// TIA Portal project "LCR 01-001" (V14)
// Atualização de hardware e software, melhorais na estrela de frasco

(* hardware
DEVICE "S7-1200 station_1"  S7-1200 Station
   slot 0: "Rack_0"  S7-1200 Rack  Rack  V1.0
   slot 1: "PLC_1"  CPU 1212C DC/DC/DC  6ES7 212-1AE40-0XB0  V4.2
   slot 3: "DQ 4x24VDC_1"  DQ4 signal board (200 kHz)  6ES7 222-1BD30-0XB0  V1.0
DEVICE "GSD device_1"  GSD.Device.PN
   slot 0: "Rack"  Rack  V1.0
   slot 0: "16DI"  16DI
   slot 0: "16DO"  16DO
   slot 0: "16DO"  16DO
   slot 0: "8DI"  8DI
   slot 0: "wago-750-375"  750-375 V02.02.xx (FW 05)  750-375  V02.02.xx (05)
      slot 0: "Big Endian (MOTOROLA), Subslot-controlled PROFIenergy"  Big Endian (MOTOROLA), Subslot-controlled PROFIenergy
      slot 1: "Interface"  Interface
         slot 1: "Port 1"  Port 1
         slot 2: "Port 2"  Port 2
   slot 1: "750-1405 16DI_1"  750-1405 16DI  750-1405
   slot 2: "750-1504 16DO_1"  750-1504 16DO  750-1504
   slot 3: "750-1504 16DO_2"  750-1504 16DO  750-1504
   slot 4: "75x-430(/0..-...) 8DI_1"  75x-430(/0..-...) 8DI  75x-430
*)

// ===== PLC "PLC_1"  CPU 1212C DC/DC/DC =====

VAR_GLOBAL   // PLC tag table "Default tag table"
   "Sensor home Platô" AT %I0.0 : Bool;
   "Sensor home Estrela" AT %I0.1 : Bool;
   "Sensor home Dosador" AT %I0.2 : Bool;
   "Sensor Limite superior Dosador" AT %I0.3 : Bool;
   "Sensor DR valvula Dosador" AT %I0.4 : Bool;
   "Sensor EQ valvula Dosador" AT %I0.5 : Bool;
   "Sensor home trans manipulador" AT %I0.6 : Bool;
   "Sensor CNT frasco dosador" AT %I0.7 : Bool;
   "Sensor CNT tampa rosqueador" AT %I1.0 : Bool;
   "Sensor canaleta de frasco" AT %I1.1 : Bool;
   "Sensor direito canaleta de tampa" AT %I1.2 : Bool;
   "Sensor esquerdo canaleta de tampa" AT %I1.3 : Bool;
   "Sensor cilindro manipulador" AT %I1.4 : Bool;
   "Sensor cilindro rosqueador" AT %I1.5 : Bool;
   "Sensor visão artificial" AT %I1.6 : Bool;
   "Sobrecarga_manipulador" AT %I1.7 : Bool;
   "Emergência" AT %I2.0 : Bool;
   "Automatico" AT %I2.1 : Bool;
   "Liga" AT %I2.2 : Bool;
   "Desliga" AT %I2.3 : Bool;
   "Reset falhas" AT %I2.4 : Bool;
   "Ativoalarmeplatô" AT %I2.5 : Bool;
   "Ativoalarmeestrela" AT %I2.6 : Bool;
   "Ativoalarmedosador" AT %I2.7 : Bool;
   "Entrada analogica" AT %IW64 : Word;
   "Sensor pressão" AT %ID200 : DWord;
   "AUX" AT %ID204 : Real;
   "CONTROLE" AT %ID208 : Real;
   "Alarme_disjunto_wago" AT %I3.0 : Bool;
   "Alvo_atingido_torque" AT %I3.1 : Bool;
   "Sensor_detector_inspeção" AT %I3.2 : Bool;
   "Sensor_CNT_manipulador" AT %I3.3 : Bool;
   "Platô_Pulse" AT %Q4.0 : Bool;
   "Platô_Direction" AT %Q4.1 : Bool;
   "Estrela_Pulse" AT %Q4.2 : Bool;
   "Estrela_Direction" AT %Q4.3 : Bool;
   "Envase_Pulse" AT %Q0.0 : Bool;
   "Envase_Direction" AT %Q0.1 : Bool;
   "Trans manipulador_Pulse" AT %Q0.2 : Bool;
   "Trans manipulador_Direction" AT %Q0.3 : Bool;
   "Smart_camera" AT %Q0.4 : Bool;
   "reservado(5)" AT %Q0.5 : Bool;
   "Gira posicinador direito tampa" AT %Q1.0 : Bool;
   "Home posicionador direito" AT %Q1.1 : Bool;
   "Gira posicionador esquerdo" AT %Q1.2 : Bool;
   "Home posicionador esquerdo" AT %Q1.3 : Bool;
   "Rosqueador aplicação tampa" AT %Q1.4 : Bool;
   "Continuo_Rosqueador" AT %Q1.5 : Bool;
   "Solenoide Rosqueador tampa" AT %Q1.6 : Bool;
   "Solenoide Manipulador tampa" AT %Q1.7 : Bool;
   "Solenoide empurrador tampa" AT %Q2.0 : Bool;
   "Solenoide valvula dosagem" AT %Q2.1 : Bool;
   "Solenoide frasco reprovado" AT %Q2.2 : Bool;
   "Válvula vacuo Pegador 1" AT %Q2.3 : Bool;
   "Válvula vacuo pegador 2" AT %Q2.4 : Bool;
   "Válvula vacuo estrela" AT %Q2.5 : Bool;
   "Válvula sopro pegador 1" AT %Q2.6 : Bool;
   "Válvula sopro pegador 2" AT %Q2.7 : Bool;
   "Válvula sopro canleta dire" AT %Q5.0 : Bool;
   "Válvula sopro canaleta esque" AT %Q5.1 : Bool;
   "Habilita alimentadores" AT %Q5.2 : Bool;
   "Alimentador de frasco" AT %Q5.3 : Bool;
   "Alimentador de tampa" AT %Q5.4 : Bool;
   "LED máquina on" AT %Q5.5 : Bool;
   "LED alarme" AT %Q5.6 : Bool;
   "LED máquina off" AT %Q5.7 : Bool;
   "Reset disjuntor eletrônico" AT %Q6.0 : Bool;
   "Reset servodrives" AT %Q6.1 : Bool;
   "Jog platô avança SV" AT %Q6.2 : Bool;
   "Jog platô recuo SV" AT %Q6.3 : Bool;
   "Jog estrela avança SV" AT %Q6.4 : Bool;
   "Jog estrela recuo SV" AT %Q6.5 : Bool;
   "Sensor_detector" AT %Q6.6 : Bool;
   "Tag_1" AT %Q6.7 : Bool;
   "System_Byte" AT %MB1 : Byte;
   "FirstScan" AT %M1.0 : Bool;
   "DiagStatusUpdate" AT %M1.1 : Bool;
   "AlwaysTRUE" AT %M1.2 : Bool;
   "AlwaysFALSE" AT %M1.3 : Bool;
   "Clock_Byte" AT %MB0 : Byte;
   "Clock_10Hz" AT %M0.0 : Bool;
   "Clock_5Hz" AT %M0.1 : Bool;
   "Clock_2.5Hz" AT %M0.2 : Bool;
   "Clock_2Hz" AT %M0.3 : Bool;
   "Clock_1.25Hz" AT %M0.4 : Bool;
   "Clock_1Hz" AT %M0.5 : Bool;
   "Clock_0.625Hz" AT %M0.6 : Bool;
   "Clock_0.5Hz" AT %M0.7 : Bool;
   "Alarme alimentador desligado" AT %M2.1 : Bool;
   "Canaletas de tampa cheia" AT %M2.2 : Bool;
   "Canaleta de tamapa vasia" AT %M2.3 : Bool;
   "Alarme falta frasco" AT %M2.4 : Bool;
   "Alarme falta tampa" AT %M2.5 : Bool;
   "Liga Máquina" AT %M2.0 : Bool;
   "Pulso  deslocamento trans" AT %M2.6 : Bool;
   "Platô em deslocamento" AT %M2.7 : Bool;
   "Platô_Alvo atingido" AT %M3.0 : Bool;
   "Estrela em deslocamento" AT %M3.1 : Bool;
   "Estrela_Alvo atingido" AT %M3.2 : Bool;
   "Envase em deslocamento" AT %M3.3 : Bool;
   "Envase_Alvo atingido" AT %M3.4 : Bool;
   "Manipulador em deslocamento" AT %M3.5 : Bool;
   "Manipulador_Alvo atingido" AT %M3.6 : Bool;
   "Falha platô" AT %M3.7 : Bool;
   "Falha etrela" AT %M4.0 : Bool;
   "Falha  envase" AT %M4.1 : Bool;
   "Falha manipu" AT %M4.2 : Bool;
   "Pulso deslocamento envase" AT %M4.3 : Bool;
   "Iniciaenvase" AT %M4.4 : Bool;
   "Iniciaenchimento" AT %M4.5 : Bool;
   "Envase_echimento alvo atingido" AT %M4.6 : Bool;
   "Envase_enchimento em deslocamento" AT %M4.7 : Bool;
   "Avança manipulador" AT %M5.0 : Bool;
   "Recuo manipulador" AT %M5.1 : Bool;
   "Set on Home platô" AT %M5.2 : Bool;
   "Set on Home estrela" AT %M5.3 : Bool;
   "Set on Home envase" AT %M5.4 : Bool;
   "Set on Home mani" AT %M5.5 : Bool;
   "Rqs_SaveReceita" AT %M6.0 : Bool;
   "Download_receita" AT %M6.1 : Bool;
   "Pulso_valavula_dosagem" AT %M6.2 : Bool;
   "Atenção" AT %M6.3 : Bool;
   "Estações_Nsincronizada" AT %M6.4 : Bool;
   "Estçoes_emhome" AT %M6.5 : Bool;
   "Bit_on" AT %M6.6 : Bool;
   "Startup_emergência" AT %M6.7 : Bool;
   "Alvo_atingidoavançoMN" AT %M7.0 : Bool;
   "Alvo_atingidorecuoMN" AT %M7.1 : Bool;
   "Deslocamento_avançoMN" AT %M7.2 : Bool;
   "Deslocamento_recuoMN" AT %M7.3 : Bool;
   "Alarme_manutenção" AT %M7.4 : Bool;
   "Status_deslocamento_rosqueador" AT %M7.5 : Bool;
   "Erro" AT %MW8 : Int;
END_VAR

TYPE "UDT_Dados_máquina"
VERSION : 0.1
   STRUCT
      Qauntidade_partida : DInt;
      Maquina_ligadahoras : DInt;
      Maquina_ligadaminutos : DInt;
      Proxima_manutenção : DInt := 0;
      Preset_manutenção : DInt;
      Salva_proximamanutenção : Bool;
   END_STRUCT;
END_TYPE

DATA_BLOCK "Start stop Machine_DB"   // DB25
{ S7_Optimized_Access := 'TRUE' }
VERSION : 0.1
// stored: InstanceOfName Start stop Machine
"Start stop Machine"
BEGIN
END_DATA_BLOCK

DATA_BLOCK "Parâmetros platô estrela"   // DB26
{ S7_Optimized_Access := 'FALSE' }
VERSION : 0.1
   VAR
      "Habilita servo drive P" : Bool;
      "Habilita Servo drive E" : Bool;
      "Habilita rampa AC/DC P" : Bool;
      "Habilita rampa AC/Dc E" : Bool;
      "Home platô" : Bool;
      "Home estrela" : Bool;
      "Jog Avanço P" : Bool;
      "Jog Recuo P" : Bool;
      "Jog avanço E" : Bool;
      "Jog recuo E" : Bool;
      "Jog avanço teste" : Bool;
      "Reset posição" : Real;
      "Jog recuo teste" : Bool;
      "Rampa aceleração" : Int;
      "Rampa desaceleração" : Int;
      "Velocidade máquina" : Int;
      "Fino home platô" : Int;
      "Fino home estrela" : Int;
      "Contador de frasco" : Int;
      Velocidadereal : Real;
      "Rampaaceleração Real" : Real;
      RampadesaceleraçãoReal : Real;
      "Fino home platô Real" : Real;
      "Fino Home estrela Real" : Real;
      "Ativa parametro" : Bool;
      "Intervalo X" : Real;
      "RampaREAL AC" : Real;
      "RampaREAL DC" : Real;
      "Home platô ON" : Bool;
      "Home estrela ON" : Bool;
      "Vacuo estrela" : Bool;
      "posição atual" : Real;
      Ganho_RPM_estrela : Real;
      Posição_atualP : Int;
      "Offset home" : Real;
      Loadparametro : Bool;
   END_VAR
BEGIN
END_DATA_BLOCK

DATA_BLOCK "Alarme_Bit"   // DB27
{ S7_Optimized_Access := 'FALSE' }
VERSION : 0.1
   VAR
      Status_sincrinizamos : Bool;
      Emergência : Bool;
      "Servo drive platõ em flha" : Bool;
      "Servo drive estrela em flha" : Bool;
      "Servo drive dosador em falha" : Bool;
      "alimentadores desligado" : Bool;
      "Alarme falta de frasco" : Bool;
      "Alrme falta de tampa" : Bool;
      "Falha instrução platô" : Bool;
      "Falha Instrução etrela" : Bool;
      "Falha instrução envase" : Bool;
      "Falha instrução manipu" : Bool;
      Falha_arcomprimido : Bool;
      Falha_Valvuladosagen : Bool;
      Falha_manipulador : Bool;
      Limite_horas : Bool;
      Sobrecarga_manipulador : Bool;
      Falha_subida_rosqueador : Bool;
      Falha_recuo_dosador : Bool;
      Falha_sensor_valvula : Bool;
   END_VAR
BEGIN
END_DATA_BLOCK

DATA_BLOCK "Parâmetros de envase"   // DB28
{ S7_Optimized_Access := 'FALSE' }
VERSION : 0.1
   VAR
      "Habilita Servo drive D" : Bool := FALSE;
      "Habilita rampa AC/DC D" : Bool := FALSE;
      "Home dosador" : Bool := FALSE;
      "Jog avanço D" : Bool := FALSE;
      "Jog recuo D" : Bool := FALSE;
      "Coreção ml" : Int := 0;
      "Rampa acelreção D" : Int := 0;
      "Rampa desaceleração D" : Int := 0;
      "Velocidade envase" : Int := 0;
      "Velocidade enchimento" : Int := 0;
      Deslocamento : Real;
      Deslocamento_1 : Real := 0.0;
      "Velocidade envase_1" : Real := 0.0;
      "Velcidade envase_2" : Real;
      Posiçãoatual : Real;
      AtivaparametrosRampa : Bool;
      "Velocidade enchimento_1" : Real;
      "Velocidade enchimento_2" : Real;
      Ramp_AC1 : Real;
      Ramp_AC2 : Real;
      Ramp_DC1 : Real;
      Ramp_DC2 : Real;
      "Home envase ON" : Bool;
      Atual_posição : Real;
      Atual_posição_scalX : Real;
      Atual_Posição_IHM : Int;
      Status_lavgem : Bool;
   END_VAR
BEGIN
END_DATA_BLOCK

DATA_BLOCK "Parâmetros rosqueador"   // DB29
{ S7_Optimized_Access := 'FALSE' }
VERSION : 0.1
   VAR
      "Desce rosqueador" : Bool;
      "Ciclo de fechamento" : Bool;
      Inter_conti : Bool;
      "Tempo deslocame_real" : Time;
      "Tempo deslocamento" : Time;
      Inicio_torque : Time;
   END_VAR
BEGIN
END_DATA_BLOCK

DATA_BLOCK "Parâmetros alimentadores_1"   // DB30
{ S7_Optimized_Access := 'FALSE' }
VERSION : 0.1
   VAR
      "Habilita frasco" : Bool;
      "Habilita tampa" : Bool;
      "ON alarme falat frasco" : Bool;
      "ON alarme falta tampa" : Bool;
      "Liga alimentadores" : Bool;
      "Retardo liga frasco" : DInt;
      "Retardo desliga frasco" : DInt;
      "Retardo liga tampa" : DInt;
      "Retardo desliga tampa" : DInt;
      "Retardo sopro D" : DInt;
      "Retardo sopro E" : DInt;
      "Retardo falta de frasco" : DInt;
      "Retardo falta de tampa" : DInt;
      Aux_realtampa : DInt;
      Aux_realfrasco : DInt;
      "Ar comprimido" : Int;
      Real_timerTampa : Int;
      Real_timerfrasco : Int;
   END_VAR
BEGIN
END_DATA_BLOCK

DATA_BLOCK "Parâmetros manipuladpor"   // DB31
{ S7_Optimized_Access := 'FALSE' }
VERSION : 0.1
   VAR
      "Habilita STR8" : Bool;
      "Habilita rampa AC/DC" : Bool;
      "Home manipulador" : Bool;
      "Jog avanço mani" : Bool;
      "Jog recuo mani" : Bool;
      "Home posici direito" : Bool;
      "Home posici esquerdo" : Bool;
      "Rampa aceleração mani" : Int;
      "Rampa desaceleração mani" : Int;
      "RPM manipulador" : Int;
      "RPM manipulador_1" : Real;
      "RPM manipulador_2" : Real;
      "Ramp AC_1" : Real;
      "Ramp AC_2" : Real;
      "Ramp DC_1" : Real;
      "Ramp DC_2" : Real;
      "ativa parametro" : Bool;
      "Posição atual_1" : Real;
      "Posição atual" : Int;
      "Home mani ON" : Bool;
      Tampa_frasco : Bool;
   END_VAR
BEGIN
END_DATA_BLOCK

DATA_BLOCK "Parâmetros de produção"   // DB32
{ S7_Optimized_Access := 'FALSE' }
VERSION : 0.1
   VAR
      "Habilita contador de lote" : Bool;
      Rejeito : Bool;
      Teste_Sensor : Bool;
      Rest_produção : Bool;
      "Peças por minuto" : DInt;
      "Total por minuto" : DInt;
      "Total por minuto_1" : Int;
      TImer_1 : Time;
      Timer_2 : Time;
      AUX_produção : Int;
   END_VAR
BEGIN
END_DATA_BLOCK

DATA_BLOCK "DB_pulso"   // DB38
{ S7_Optimized_Access := 'TRUE' }
VERSION : 0.1
   VAR
      Manual : Bool;
      Pulso_PL_ES : Array[0..12] of Bool;
      Pulso_EV : Array[0..20] of Bool;
      Pulso_MN : Array[0..25] of Bool;
      Pulso_RQ : Array[0..10] of Bool;
      Pulso_ALM : Array[0..20] of Bool;
      Pulso_receita : Array[0..5] of Bool;
      Pulso_alarme : Array[0..20] of Bool;
      Controle_produção : Array[0..20] of Bool;
      Startup : Array[0..20] of Bool;
      UDT_máquina : Array[0..5] of Bool;
   END_VAR
BEGIN
END_DATA_BLOCK

DATA_BLOCK "Comando transmissão_DB"   // DB43
{ S7_Optimized_Access := 'TRUE' }
VERSION : 0.1
// stored: InstanceOfName Comando transmissão
"Comando transmissão"
BEGIN
END_DATA_BLOCK

DATA_BLOCK "Comando valvula dosador_DB"   // DB48
{ S7_Optimized_Access := 'TRUE' }
VERSION : 0.1
// stored: InstanceOfName Comando valvula dosador
"Comando valvula dosador"
BEGIN
END_DATA_BLOCK

DATA_BLOCK "Controle manipulador_DB"   // DB51
{ S7_Optimized_Access := 'TRUE' }
VERSION : 0.1
// stored: InstanceOfName Controle manipulador
"Controle manipulador"
BEGIN
END_DATA_BLOCK

DATA_BLOCK "DB_UDT_dadosMáqquin"   // DB53
{ S7_Optimized_Access := 'FALSE' }
VERSION : 0.1
   VAR
      Plc_DT_atual : DTL;
      Retorvalor : Int;
      Máquina : Array[0..0] of "UDT_Dados_máquina";
      Aux_preset : Int;
      Aux_horas : Int;
      Aux_minuto : Int;
      Aux_partida : Int;
   END_VAR
BEGIN
END_DATA_BLOCK

DATA_BLOCK "DB_Receitas"   // DB55
{ S7_Optimized_Access := 'FALSE' }
VERSION : 0.1
   VAR
      Receita : Array[0..20] of Word;
      Rqs_DownloadReceita : Bool;
      Rqs_SaveReceita : Bool;
   END_VAR
BEGIN
END_DATA_BLOCK

DATA_BLOCK "Parâmetros_IHM"   // DB56
{ S7_Optimized_Access := 'FALSE' }
VERSION : 0.1
   VAR
      Int_1 : Int;
      Int_2 : Int;
      Int_3 : Int;
      Int_4 : Int;
      Int_5 : Int;
      Int_6 : Int;
      Int_7 : Int;
      Int_8 : Int;
      Int_9 : Int;
      Int_10 : Int;
      Int_11 : Int;
      Int_12 : Int;
      Int_13 : Int;
      Int_14 : Int;
      Int_15 : Int;
      Int_16 : Int;
      Int_17 : Int;
      Int_18 : Int;
      Int_19 : Int;
      Int_20 : Int;
      Int_21 : Int;
      Int_22 : Int;
      Int_23 : Int;
      Int_24 : Int;
      Int_25 : Int;
      Int_26 : Int;
      Int_27 : Int;
      Int_28 : Int;
      Int_29 : Int;
      Int_30 : Int;
      Int_31 : Int;
      Int_32 : Int;
      Int_33 : Int;
      Int_34 : Int;
      Int_35 : Int;
      Int_36 : Int;
      Int_37 : Int;
      Int_38 : Int;
      Int_39 : Int;
      Int_40 : Int;
      DBW_0 : Word;
   END_VAR
BEGIN
END_DATA_BLOCK

DATA_BLOCK "Parâmetros_BooL_IHM"   // DB57
{ S7_Optimized_Access := 'FALSE' }
VERSION : 0.1
   VAR
      St001 : Bool;
      St002 : Bool;
      St003 : Bool;
      St004 : Bool;
      St005 : Bool;
      St006 : Bool;
      St007 : Bool;
      St008 : Bool;
      St009 : Bool;
      St010 : Bool;
      St011 : Bool;
      St012 : Bool;
      St013 : Bool;
      St014 : Bool;
      St015 : Bool;
      St016 : Bool;
      St017 : Bool;
      St018 : Bool;
      St019 : Bool;
      St020 : Bool;
      Status_W0 : Int;
      Status_W1 : Int;
   END_VAR
BEGIN
END_DATA_BLOCK

DATA_BLOCK "Rosqueador_tampa_DB"   // DB59
{ S7_Optimized_Access := 'TRUE' }
VERSION : 0.1
// stored: InstanceOfName Rosqueador_tampa
"Rosqueador_tampa"
BEGIN
END_DATA_BLOCK

DATA_BLOCK "Alarme_mensagen"   // DB60
{ S7_Optimized_Access := 'FALSE' }
VERSION : 0.1
   VAR
      Mensagen_1 : Array[0..15] of Word;
   END_VAR
BEGIN
END_DATA_BLOCK

DATA_BLOCK "DB_Startup"   // DB68
{ S7_Optimized_Access := 'TRUE' }
VERSION : 0.1
   VAR
      Stsrtup : Array[0..10] of Bool;
   END_VAR
BEGIN
END_DATA_BLOCK

DATA_BLOCK "Presença"   // DB72
{ S7_Optimized_Access := 'FALSE' }
VERSION : 0.1
   VAR
      Presenca_08 : Bool;
      Presenca_09 : Bool;
      Presenca_10 : Bool;
      Presenca_11 : Bool;
      Presenca_12 : Bool;
      Presenca_13 : Bool;
      Presenca_14 : Bool;
      Presenca_15 : Bool;
      Presenca_00 : Bool;
      Presenca_01 : Bool;
      Presenca_02 : Bool;
      Presenca_03 : Bool;
      Presenca_04 : Bool;
      Presenca_05 : Bool;
      Presenca_06 : Bool;
      Presenca_07 : Bool;
   END_VAR
BEGIN
END_DATA_BLOCK

// folder: System blocks/Program resources

DATA_BLOCK "IEC_Timer_0_DB"   // DB33
{ S7_Optimized_Access := 'TRUE' }
AUTHOR : Simatic
FAMILY : IEC
NAME : IEC_TMR
VERSION : 1.0
// stored: InstanceOfName IEC_TIMER
"IEC_TIMER"
BEGIN
END_DATA_BLOCK

DATA_BLOCK "IEC_Timer_0_DB_1"   // DB34
{ S7_Optimized_Access := 'TRUE' }
AUTHOR : Simatic
FAMILY : IEC
NAME : IEC_TMR
VERSION : 1.0
// stored: InstanceOfName IEC_TIMER
"IEC_TIMER"
BEGIN
END_DATA_BLOCK

DATA_BLOCK "IEC_Timer_0_DB_2"   // DB35
{ S7_Optimized_Access := 'TRUE' }
AUTHOR : Simatic
FAMILY : IEC
NAME : IEC_TMR
VERSION : 1.0
// stored: InstanceOfName IEC_TIMER
"IEC_TIMER"
BEGIN
END_DATA_BLOCK

DATA_BLOCK "IEC_Timer_0_DB_3"   // DB36
{ S7_Optimized_Access := 'TRUE' }
AUTHOR : Simatic
FAMILY : IEC
NAME : IEC_TMR
VERSION : 1.0
// stored: InstanceOfName IEC_TIMER
"IEC_TIMER"
BEGIN
END_DATA_BLOCK

DATA_BLOCK "IEC_Timer_0_DB_4"   // DB37
{ S7_Optimized_Access := 'TRUE' }
AUTHOR : Simatic
FAMILY : IEC
NAME : IEC_TMR
VERSION : 1.0
// stored: InstanceOfName IEC_TIMER
"IEC_TIMER"
BEGIN
END_DATA_BLOCK

DATA_BLOCK "IEC_Timer_0_DB_5"   // DB39
{ S7_Optimized_Access := 'TRUE' }
AUTHOR : Simatic
FAMILY : IEC
NAME : IEC_TMR
VERSION : 1.0
// stored: InstanceOfName IEC_TIMER
"IEC_TIMER"
BEGIN
END_DATA_BLOCK

DATA_BLOCK "IEC_Timer_0_DB_6"   // DB40
{ S7_Optimized_Access := 'TRUE' }
AUTHOR : Simatic
FAMILY : IEC
NAME : IEC_TMR
VERSION : 1.0
// stored: InstanceOfName IEC_TIMER
"IEC_TIMER"
BEGIN
END_DATA_BLOCK

DATA_BLOCK "IEC_Timer_0_DB_7"   // DB41
{ S7_Optimized_Access := 'TRUE' }
AUTHOR : Simatic
FAMILY : IEC
NAME : IEC_TMR
VERSION : 1.0
// stored: InstanceOfName IEC_TIMER
"IEC_TIMER"
BEGIN
END_DATA_BLOCK

DATA_BLOCK "IEC_Timer_0_DB_8"   // DB42
{ S7_Optimized_Access := 'TRUE' }
AUTHOR : Simatic
FAMILY : IEC
NAME : IEC_TMR
VERSION : 1.0
// stored: InstanceOfName IEC_TIMER
"IEC_TIMER"
BEGIN
END_DATA_BLOCK

DATA_BLOCK "IEC_Timer_0_DB_9"   // DB50
{ S7_Optimized_Access := 'TRUE' }
AUTHOR : Simatic
FAMILY : IEC
NAME : IEC_TMR
VERSION : 1.0
// stored: InstanceOfName IEC_TIMER
"IEC_TIMER"
BEGIN
END_DATA_BLOCK

DATA_BLOCK "IEC_Timer_0_DB_10"   // DB61
{ S7_Optimized_Access := 'TRUE' }
AUTHOR : Simatic
FAMILY : IEC
NAME : IEC_TMR
VERSION : 1.0
// stored: InstanceOfName IEC_TIMER
"IEC_TIMER"
BEGIN
END_DATA_BLOCK

DATA_BLOCK "IEC_Timer_0_DB_11"   // DB62
{ S7_Optimized_Access := 'TRUE' }
AUTHOR : Simatic
FAMILY : IEC
NAME : IEC_TMR
VERSION : 1.0
// stored: InstanceOfName IEC_TIMER
"IEC_TIMER"
BEGIN
END_DATA_BLOCK

DATA_BLOCK "IEC_Timer_0_DB_12"   // DB63
{ S7_Optimized_Access := 'TRUE' }
AUTHOR : Simatic
FAMILY : IEC
NAME : IEC_TMR
VERSION : 1.0
// stored: InstanceOfName IEC_TIMER
"IEC_TIMER"
BEGIN
END_DATA_BLOCK

DATA_BLOCK "IEC_Timer_0_DB_19"   // DB64
{ S7_Optimized_Access := 'TRUE' }
AUTHOR : Simatic
FAMILY : IEC
NAME : IEC_TMR
VERSION : 1.0
// stored: InstanceOfName IEC_TIMER
"IEC_TIMER"
BEGIN
END_DATA_BLOCK

DATA_BLOCK "IEC_Timer_0_DB_13"   // DB65
{ S7_Optimized_Access := 'TRUE' }
AUTHOR : Simatic
FAMILY : IEC
NAME : IEC_TMR
VERSION : 1.0
// stored: InstanceOfName IEC_TIMER
"IEC_TIMER"
BEGIN
END_DATA_BLOCK

DATA_BLOCK "IEC_Timer_0_DB_14"   // DB66
{ S7_Optimized_Access := 'TRUE' }
AUTHOR : Simatic
FAMILY : IEC
NAME : IEC_TMR
VERSION : 1.0
// stored: InstanceOfName IEC_TIMER
"IEC_TIMER"
BEGIN
END_DATA_BLOCK

DATA_BLOCK "IEC_Timer_0_DB_15"   // DB67
{ S7_Optimized_Access := 'TRUE' }
AUTHOR : Simatic
FAMILY : IEC
NAME : IEC_TMR
VERSION : 1.0
// stored: InstanceOfName IEC_TIMER
"IEC_TIMER"
BEGIN
END_DATA_BLOCK

DATA_BLOCK "IEC_Timer_0_DB_16"   // DB69
{ S7_Optimized_Access := 'TRUE' }
AUTHOR : Simatic
FAMILY : IEC
NAME : IEC_TMR
VERSION : 1.0
// stored: InstanceOfName IEC_TIMER
"IEC_TIMER"
BEGIN
END_DATA_BLOCK

DATA_BLOCK "IEC_Timer_0_DB_17"   // DB70
{ S7_Optimized_Access := 'TRUE' }
AUTHOR : Simatic
FAMILY : IEC
NAME : IEC_TMR
VERSION : 1.0
// stored: InstanceOfName IEC_TIMER
"IEC_TIMER"
BEGIN
END_DATA_BLOCK

DATA_BLOCK "IEC_Timer_0_DB_18"   // DB71
{ S7_Optimized_Access := 'TRUE' }
AUTHOR : Simatic
FAMILY : IEC
NAME : IEC_TMR
VERSION : 1.0
// stored: InstanceOfName IEC_TIMER
"IEC_TIMER"
BEGIN
END_DATA_BLOCK

// folder: (top level)

DATA_BLOCK "Platô"   // DB2, Motion_DB
{ S7_Optimized_Access := 'TRUE' }
AUTHOR : SIMATIC
FAMILY : BasicMC
NAME : TO_PosAx
VERSION : 5.0
// stored: InstanceOfName TO_PositioningAxis
"TO_PositioningAxis"
BEGIN
   // Axis.LengthUnitNormalized.Distance = 1005
   // Axis.PositionLimitsMin_AddressCU = %I0.0
   // Axis.DirectionOutputEnabledCU = TRUE
   // Axis.PassiveHomingReferencePointSwitch_AddressCU = %I0.0
   // Axis.HomingReferencePointSwitch_AddressCU = %I0.0
   // Axis.OnlinePtoModeCUEnumValue = PTO (pulse A and direction B)
   // Axis.OnlinePtoModeCU = 16#0000_0002
   // Axis.SelectedChannel2EnumCU = %Q4.1
   // Axis.SelectedChannel1EnumCU = %Q4.0
   // Pulse.MinDeltaDeltaFrequencyCU = 0.004
   // Pulse.MaxDeltaDeltaFrequencyCU = 1.0E+10
   // Pulse.MinDeltaFrequencyCU = 0.005
   // Pulse.MaxDeltaFrequencyCU = 9.5E+9
   // Pulse.MinFrequencyCU = 1.0
   // Pulse.MaxFrequencyCU = 200000.0
   // Pulse.OutputSourceCU = 16#0000_0001
   // Axis.SelectPTO = 0
   // Axis.LengthUnit.LastDistance = 1005
END_DATA_BLOCK

DATA_BLOCK "Estrela"   // DB3, Motion_DB
{ S7_Optimized_Access := 'TRUE' }
AUTHOR : SIMATIC
FAMILY : BasicMC
NAME : TO_PosAx
VERSION : 5.0
// stored: InstanceOfName TO_PositioningAxis
"TO_PositioningAxis"
BEGIN
   // Axis.PositionLimitsMin_AddressCU = %I0.1
   // Axis.PassiveHomingReferencePointSwitch_AddressCU = %I0.1
   // Axis.HomingReferencePointSwitch_AddressCU = %I0.1
   // Axis.LengthUnitNormalized.Distance = 1005
   // Axis.DirectionOutputEnabledCU = TRUE
   // Axis.OnlinePtoModeCUEnumValue = PTO (pulse A and direction B)
   // Axis.OnlinePtoModeCU = 16#0000_0002
   // Axis.SelectedChannel2EnumCU = %Q4.3
   // Axis.SelectedChannel1EnumCU = %Q4.2
   // Pulse.MinDeltaDeltaFrequencyCU = 0.004
   // Pulse.MaxDeltaDeltaFrequencyCU = 1.0E+10
   // Pulse.MinDeltaFrequencyCU = 0.005
   // Pulse.MaxDeltaFrequencyCU = 9.5E+9
   // Pulse.MinFrequencyCU = 1.0
   // Pulse.MaxFrequencyCU = 200000.0
   // Pulse.OutputSourceCU = 16#0000_0001
   // Axis.SelectPTO = 1
   // Axis.OnlinePtoIndexCU = 1
   // Axis.LengthUnit.LastDistance = 1005
END_DATA_BLOCK

DATA_BLOCK "Envase"   // DB4, Motion_DB
{ S7_Optimized_Access := 'TRUE' }
AUTHOR : SIMATIC
FAMILY : BasicMC
NAME : TO_PosAx
VERSION : 5.0
// stored: InstanceOfName TO_PositioningAxis
"TO_PositioningAxis"
BEGIN
   // Axis.PositionLimitsMax_AddressCU = %I0.3
   // Axis.PositionLimitsMin_AddressCU = %I0.2
   // Axis.PassiveHomingReferencePointSwitch_AddressCU = %I0.2
   // Axis.HomingReferencePointSwitch_AddressCU = %I0.2
   // Axis.LengthUnitNormalized.Distance = 1005
   // Axis.DirectionOutputEnabledCU = TRUE
   // Axis.OnlinePtoModeCUEnumValue = PTO (pulse A and direction B)
   // Axis.OnlinePtoModeCU = 16#0000_0002
   // Axis.SelectedChannel2EnumCU = %Q0.1
   // Axis.SelectedChannel1EnumCU = %Q0.0
   // Pulse.MinDeltaDeltaFrequencyCU = 0.004
   // Pulse.MaxDeltaDeltaFrequencyCU = 1.0E+10
   // Pulse.MinDeltaFrequencyCU = 0.005
   // Pulse.MaxDeltaFrequencyCU = 9.5E+9
   // Pulse.MinFrequencyCU = 1.0
   // Pulse.MaxFrequencyCU = 100000.0
   // Pulse.OutputSourceCU = 16#0000_0000
   // Axis.SelectPTO = 2
   // Axis.OnlinePtoIndexCU = 2
   // Axis.LengthUnit.LastDistance = 1005
END_DATA_BLOCK

DATA_BLOCK "Trans manipulador"   // DB5, Motion_DB
{ S7_Optimized_Access := 'TRUE' }
AUTHOR : SIMATIC
FAMILY : BasicMC
NAME : TO_PosAx
VERSION : 5.0
// stored: InstanceOfName TO_PositioningAxis
"TO_PositioningAxis"
BEGIN
   // Axis.PositionLimitsMax_AddressCU = %I0.6
   // Axis.PassiveHomingReferencePointSwitch_AddressCU = %I0.6
   // Axis.HomingReferencePointSwitch_AddressCU = %I0.6
   // Axis.LengthUnitNormalized.Distance = 1005
   // Axis.SelectedChannel2EnumCU = %Q0.3
   // Axis.SelectedChannel1EnumCU = %Q0.2
   // Axis.DirectionOutputEnabledCU = TRUE
   // Axis.OnlinePtoModeCUEnumValue = PTO (pulse A and direction B)
   // Axis.OnlinePtoModeCU = 16#0000_0002
   // Pulse.MinDeltaDeltaFrequencyCU = 0.004
   // Pulse.MaxDeltaDeltaFrequencyCU = 1.0E+10
   // Pulse.MinDeltaFrequencyCU = 0.005
   // Pulse.MaxDeltaFrequencyCU = 9.5E+9
   // Pulse.MinFrequencyCU = 1.0
   // Pulse.MaxFrequencyCU = 100000.0
   // Pulse.OutputSourceCU = 16#0000_0000
   // Axis.SelectPTO = 3
   // Axis.OnlinePtoIndexCU = 3
   // Axis.LengthUnit.LastDistance = 1005
END_DATA_BLOCK

FUNCTION_BLOCK "Start stop Machine"   // FB1, LAD
{ S7_Optimized_Access := 'TRUE' }
VERSION : 0.1
   VAR_INPUT
      Emergência : Bool;
      Automatico : Bool;
      Start : Bool;
      Stop : Bool;
      "Timer" : Time;
      Alarmeati_W0 : Word;
      Alarmeati_W1 : Word;
      Alarmeati_W2 : Word;
   END_VAR
   VAR_OUTPUT
      Machine_ON : Bool;
      LEDstart : Bool;
      LEDalarme : Bool;
      LEDstop : Bool;
   END_VAR
   VAR
      Statusalarme : Bool;
      Statusmachine : Bool;
      Pulso : Bool;
      IEC_Timer_0_Instance : TON_TIME;
   END_VAR
BEGIN

REGION Network 1: Habilita Máquina pronta
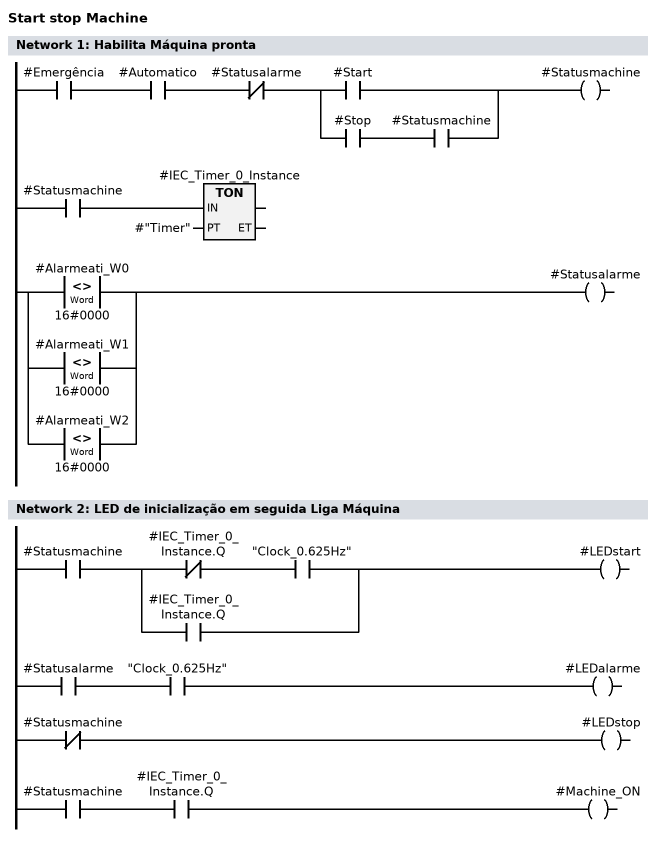
   #Statusmachine := #Emergência AND #Automatico AND NOT #Statusalarme AND (#Start OR (#Stop AND #Statusmachine));
   #IEC_Timer_0_Instance(IN := #Statusmachine, PT := #"Timer");   // TON
   #Statusalarme := (#Alarmeati_W0 <> 16#0000) OR (#Alarmeati_W1 <> 16#0000) OR (#Alarmeati_W2 <> 16#0000);
END_REGION

REGION Network 2: LED de inicialização em seguida Liga Máquina
   RUNG wire#powerrail
      Contact( #Statusmachine )
      wire#w1
      I_Contact( #IEC_Timer_0_Instance.Q )
      Contact( "Clock_0.625Hz" )
      wire#w2
      Coil( #LEDstart )
   END_RUNG
   RUNG wire#w1
      Contact( #IEC_Timer_0_Instance.Q )
   END_RUNG wire#w2
   RUNG wire#powerrail
      Contact( #Statusalarme )
      Contact( "Clock_0.625Hz" )
      Coil( #LEDalarme )
   END_RUNG
   RUNG wire#powerrail
      I_Contact( #Statusmachine )
      Coil( #LEDstop )
   END_RUNG
   RUNG wire#powerrail
      Contact( #Statusmachine )
      Contact( #IEC_Timer_0_Instance.Q )
      Coil( #Machine_ON )
   END_RUNG
   // the same network as SCL:
   #LEDstart := #Statusmachine AND ((NOT #IEC_Timer_0_Instance.Q AND "Clock_0.625Hz") OR #IEC_Timer_0_Instance.Q);
   #LEDalarme := #Statusalarme AND "Clock_0.625Hz";
   #LEDstop := NOT #Statusmachine;
   #Machine_ON := #Statusmachine AND #IEC_Timer_0_Instance.Q;
END_REGION
END_FUNCTION_BLOCK

FUNCTION_BLOCK "Comando transmissão"   // FB2, LAD
{ S7_Optimized_Access := 'TRUE' }
VERSION : 0.1
   VAR_INPUT
      "Habilita comando" : Bool;
      "Status deslocamento P" : Bool := false;
      "Status deslocamento E" : Bool;
      "Status deslocamento envase" : Bool;
      Pulsofrasco : Bool;
      Alvoatingido : Bool;
      Alvoatingido_platô : Bool;
      Fimenvase : Bool;
      Vacuo_Inte_cont : Bool;
   END_VAR
   VAR_OUTPUT
      Pulso_transmissão : Bool;
      Pulso_envase : Bool;
      Vácuo_estrela : Bool;
   END_VAR
   VAR
      Comandorodar : Bool;
      Envasehabilitado : Bool;
      Status_vacuo_estrela : Bool;
      IEC_Timer_0_Instance : TON_TIME;
   END_VAR
   VAR_TEMP   // added for the SCL form of the ladder/FBD networks
      _w1 : Bool;
      _w2 : Bool;
      _w3 : Bool;
      _w4 : Bool;
      _w5 : Bool;
      _w6 : Bool;
      _w7 : Bool;
   END_VAR
BEGIN

REGION Network 1: Habilita comando de transmissão
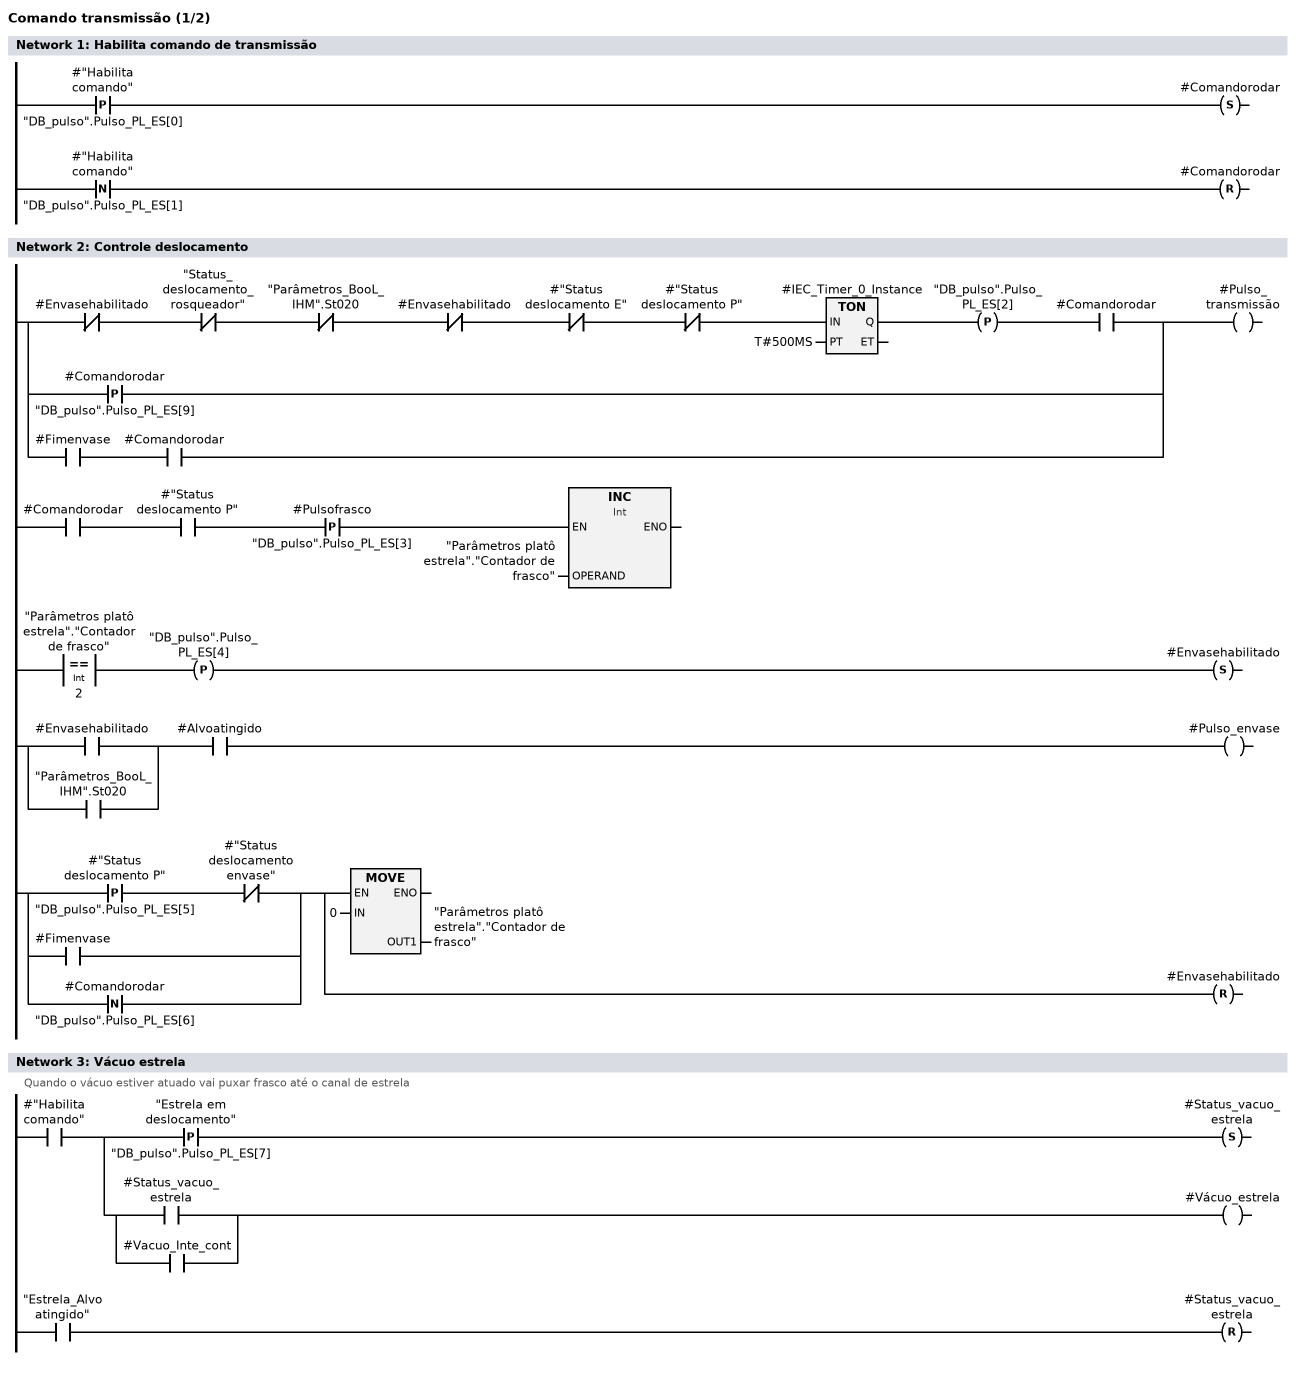
   RUNG wire#powerrail
      P_Contact(operand := #"Habilita comando", bit := "DB_pulso".Pulso_PL_ES[0])
      S_Coil( #Comandorodar )
   END_RUNG
   RUNG wire#powerrail
      N_Contact(operand := #"Habilita comando", bit := "DB_pulso".Pulso_PL_ES[1])
      R_Coil( #Comandorodar )
   END_RUNG
   // the same network as SCL:
   #_w1 := #"Habilita comando" AND NOT "DB_pulso".Pulso_PL_ES[0];   // rising edge of #"Habilita comando"
   "DB_pulso".Pulso_PL_ES[0] := #"Habilita comando";
   IF #_w1 THEN #Comandorodar := TRUE; END_IF;
   #_w2 := NOT #"Habilita comando" AND "DB_pulso".Pulso_PL_ES[1];   // falling edge of #"Habilita comando"
   "DB_pulso".Pulso_PL_ES[1] := #"Habilita comando";
   IF #_w2 THEN #Comandorodar := FALSE; END_IF;
END_REGION

REGION Network 2: Controle deslocamento
   #IEC_Timer_0_Instance(IN := NOT #Envasehabilitado AND NOT "Status_deslocamento_rosqueador" AND NOT "Parâmetros_BooL_IHM".St020 AND NOT #Envasehabilitado AND NOT #"Status deslocamento E" AND NOT #"Status deslocamento P",   // TON
                         PT := T#500MS);
   #_w1 := #IEC_Timer_0_Instance.Q AND NOT "DB_pulso".Pulso_PL_ES[2];   // rising edge
   "DB_pulso".Pulso_PL_ES[2] := #IEC_Timer_0_Instance.Q;
   #_w2 := #Comandorodar AND NOT "DB_pulso".Pulso_PL_ES[9];   // rising edge of #Comandorodar
   "DB_pulso".Pulso_PL_ES[9] := #Comandorodar;
   #Pulso_transmissão := (#_w1 AND #Comandorodar) OR #_w2 OR (#Fimenvase AND #Comandorodar);
   #_w3 := #Comandorodar AND #"Status deslocamento P" AND #Pulsofrasco AND NOT "DB_pulso".Pulso_PL_ES[3];   // rising edge of #Pulsofrasco
   "DB_pulso".Pulso_PL_ES[3] := #Pulsofrasco;
   IF #_w3 THEN
       "Parâmetros platô estrela"."Contador de frasco" := "Parâmetros platô estrela"."Contador de frasco" + 1;
   END_IF;
   #_w4 := "Parâmetros platô estrela"."Contador de frasco" = 2;
   #_w5 := #_w4 AND NOT "DB_pulso".Pulso_PL_ES[4];   // rising edge
   "DB_pulso".Pulso_PL_ES[4] := #_w4;
   IF #_w5 THEN #Envasehabilitado := TRUE; END_IF;
   #Pulso_envase := (#Envasehabilitado OR "Parâmetros_BooL_IHM".St020) AND #Alvoatingido;
   #_w6 := #"Status deslocamento P" AND NOT "DB_pulso".Pulso_PL_ES[5];   // rising edge of #"Status deslocamento P"
   "DB_pulso".Pulso_PL_ES[5] := #"Status deslocamento P";
   #_w7 := NOT #Comandorodar AND "DB_pulso".Pulso_PL_ES[6];   // falling edge of #Comandorodar
   "DB_pulso".Pulso_PL_ES[6] := #Comandorodar;
   IF (#_w6 AND NOT #"Status deslocamento envase") OR #Fimenvase OR #_w7 THEN
       "Parâmetros platô estrela"."Contador de frasco" := 0;
       #Envasehabilitado := FALSE;
   END_IF;
END_REGION

REGION Network 3: Vácuo estrela
   // Quando o vácuo estiver atuado vai puxar frasco até o canal de estrela
   RUNG wire#powerrail
      Contact( #"Habilita comando" )
      wire#w1
      P_Contact(operand := "Estrela em deslocamento", bit := "DB_pulso".Pulso_PL_ES[7])
      S_Coil( #Status_vacuo_estrela )
   END_RUNG
   RUNG wire#w1
      Contact( #Status_vacuo_estrela )
      wire#w2
      Coil( #Vácuo_estrela )
   END_RUNG
   RUNG wire#w1
      Contact( #Vacuo_Inte_cont )
   END_RUNG wire#w2
   RUNG wire#powerrail
      Contact( "Estrela_Alvo atingido" )
      R_Coil( #Status_vacuo_estrela )
   END_RUNG
   // the same network as SCL:
   #_w1 := #"Habilita comando" AND "Estrela em deslocamento" AND NOT "DB_pulso".Pulso_PL_ES[7];   // rising edge of "Estrela em deslocamento"
   "DB_pulso".Pulso_PL_ES[7] := "Estrela em deslocamento";
   IF #_w1 THEN #Status_vacuo_estrela := TRUE; END_IF;
   #Vácuo_estrela := #"Habilita comando" AND (#Status_vacuo_estrela OR #Vacuo_Inte_cont);
   IF "Estrela_Alvo atingido" THEN #Status_vacuo_estrela := FALSE; END_IF;
END_REGION

REGION Network 4: Satatus deslocamento
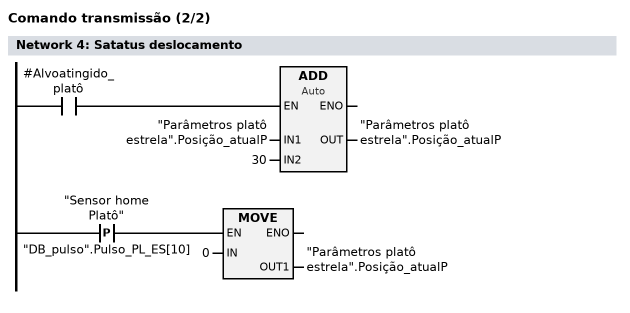
   RUNG wire#powerrail
      Contact( #Alvoatingido_platô )
      Add(in1 := "Parâmetros platô estrela".Posição_atualP, in2 := 30, out => "Parâmetros platô estrela".Posição_atualP)
   END_RUNG
   RUNG wire#powerrail
      P_Contact(operand := "Sensor home Platô", bit := "DB_pulso".Pulso_PL_ES[10])
      Move(in := 0, out1 => "Parâmetros platô estrela".Posição_atualP)
   END_RUNG
   // the same network as SCL:
   IF #Alvoatingido_platô THEN
       "Parâmetros platô estrela".Posição_atualP := "Parâmetros platô estrela".Posição_atualP + 30;
   END_IF;
   #_w1 := "Sensor home Platô" AND NOT "DB_pulso".Pulso_PL_ES[10];   // rising edge of "Sensor home Platô"
   "DB_pulso".Pulso_PL_ES[10] := "Sensor home Platô";
   IF #_w1 THEN "Parâmetros platô estrela".Posição_atualP := 0; END_IF;
END_REGION
END_FUNCTION_BLOCK

FUNCTION_BLOCK "Comando valvula dosador"   // FB3, LAD
{ S7_Optimized_Access := 'TRUE' }
VERSION : 0.1
   VAR_INPUT
      Habilitacomando : Bool;
      Envase : Bool;
      Fimenvase : Bool;
      Fimenchimento : Bool;
      Habilita_lavagem : Bool;
   END_VAR
   VAR_OUTPUT
      Valvuladosagem : Bool;
      Deslocamentoenvase : Bool;
      Deslocamentoenchimento : Bool;
      Status_lavagem : Bool;
   END_VAR
   VAR
      Comandorodar : Bool;
      Comandoenvase : Bool;
      Envasando : Bool;
      Enchendo : Bool;
      Status_valvula : Bool;
      Comando_lavagem : Bool;
      Reciclo_lavagem : Bool;
      IEC_Timer_0_Instance : TON_TIME;
      IEC_Timer_0_Instance_1 : TON_TIME;
   END_VAR
   VAR_TEMP   // added for the SCL form of the ladder/FBD networks
      _w1 : Bool;
      _w2 : Bool;
      _w3 : Bool;
      _w4 : Bool;
      _w5 : Bool;
   END_VAR
BEGIN

REGION Network 1: Habilita comando transmissão e envase continuo
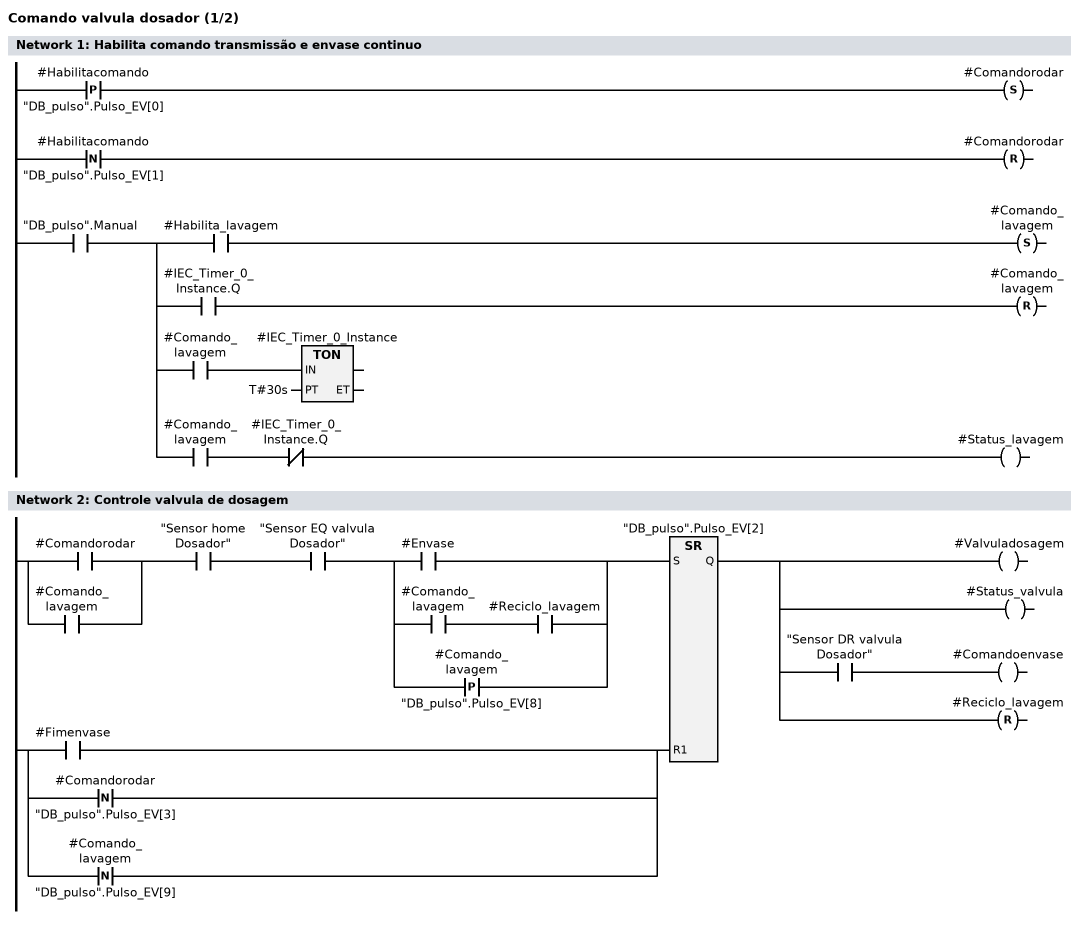
   #_w1 := #Habilitacomando AND NOT "DB_pulso".Pulso_EV[0];   // rising edge of #Habilitacomando
   "DB_pulso".Pulso_EV[0] := #Habilitacomando;
   IF #_w1 THEN #Comandorodar := TRUE; END_IF;
   #_w2 := NOT #Habilitacomando AND "DB_pulso".Pulso_EV[1];   // falling edge of #Habilitacomando
   "DB_pulso".Pulso_EV[1] := #Habilitacomando;
   IF #_w2 THEN #Comandorodar := FALSE; END_IF;
   IF "DB_pulso".Manual AND #Habilita_lavagem THEN #Comando_lavagem := TRUE; END_IF;
   IF "DB_pulso".Manual AND #IEC_Timer_0_Instance.Q THEN #Comando_lavagem := FALSE; END_IF;
   #IEC_Timer_0_Instance(IN := "DB_pulso".Manual AND #Comando_lavagem, PT := T#30s);   // TON
   #Status_lavagem := "DB_pulso".Manual AND #Comando_lavagem AND NOT #IEC_Timer_0_Instance.Q;
END_REGION

REGION Network 2: Controle valvula de dosagem
   RUNG wire#powerrail
      Contact( #Comandorodar )
      wire#w1
      Contact( "Sensor home Dosador" )
      Contact( "Sensor EQ valvula Dosador" )
      wire#w2
      Contact( #Envase )
      wire#w3
      S_SR(operand := "DB_pulso".Pulso_EV[2], r1 := wire#w4)
      wire#w5
      Coil( #Valvuladosagem )
   END_RUNG
   RUNG wire#powerrail
      Contact( #Comando_lavagem )
   END_RUNG wire#w1
   RUNG wire#w2
      Contact( #Comando_lavagem )
      Contact( #Reciclo_lavagem )
   END_RUNG wire#w3
   RUNG wire#w2
      P_Contact(operand := #Comando_lavagem, bit := "DB_pulso".Pulso_EV[8])
   END_RUNG wire#w3
   RUNG wire#powerrail
      Contact( #Fimenvase )
   END_RUNG wire#w4
   RUNG wire#powerrail
      N_Contact(operand := #Comandorodar, bit := "DB_pulso".Pulso_EV[3])
   END_RUNG wire#w4
   RUNG wire#powerrail
      N_Contact(operand := #Comando_lavagem, bit := "DB_pulso".Pulso_EV[9])
   END_RUNG wire#w4
   RUNG wire#w5
      Coil( #Status_valvula )
   END_RUNG
   RUNG wire#w5
      Contact( "Sensor DR valvula Dosador" )
      Coil( #Comandoenvase )
   END_RUNG
   RUNG wire#w5
      R_Coil( #Reciclo_lavagem )
   END_RUNG
   // the same network as SCL:
   #_w1 := (#Comandorodar OR #Comando_lavagem) AND "Sensor home Dosador" AND "Sensor EQ valvula Dosador" AND #Comando_lavagem AND NOT "DB_pulso".Pulso_EV[8];   // rising edge of #Comando_lavagem
   "DB_pulso".Pulso_EV[8] := #Comando_lavagem;
   #_w2 := NOT #Comandorodar AND "DB_pulso".Pulso_EV[3];   // falling edge of #Comandorodar
   "DB_pulso".Pulso_EV[3] := #Comandorodar;
   #_w3 := NOT #Comando_lavagem AND "DB_pulso".Pulso_EV[9];   // falling edge of #Comando_lavagem
   "DB_pulso".Pulso_EV[9] := #Comando_lavagem;
   IF ((#Comandorodar OR #Comando_lavagem) AND "Sensor home Dosador" AND "Sensor EQ valvula Dosador" AND (#Envase OR (#Comando_lavagem AND #Reciclo_lavagem))) OR #_w1 THEN
       "DB_pulso".Pulso_EV[2] := TRUE;   // SR flip-flop
   END_IF;
   IF #Fimenvase OR #_w2 OR #_w3 THEN "DB_pulso".Pulso_EV[2] := FALSE; END_IF;
   #Valvuladosagem := "DB_pulso".Pulso_EV[2];
   #Status_valvula := "DB_pulso".Pulso_EV[2];
   #Comandoenvase := "DB_pulso".Pulso_EV[2] AND "Sensor DR valvula Dosador";
   IF "DB_pulso".Pulso_EV[2] THEN #Reciclo_lavagem := FALSE; END_IF;
END_REGION

REGION Network 3: Deslocamento envase
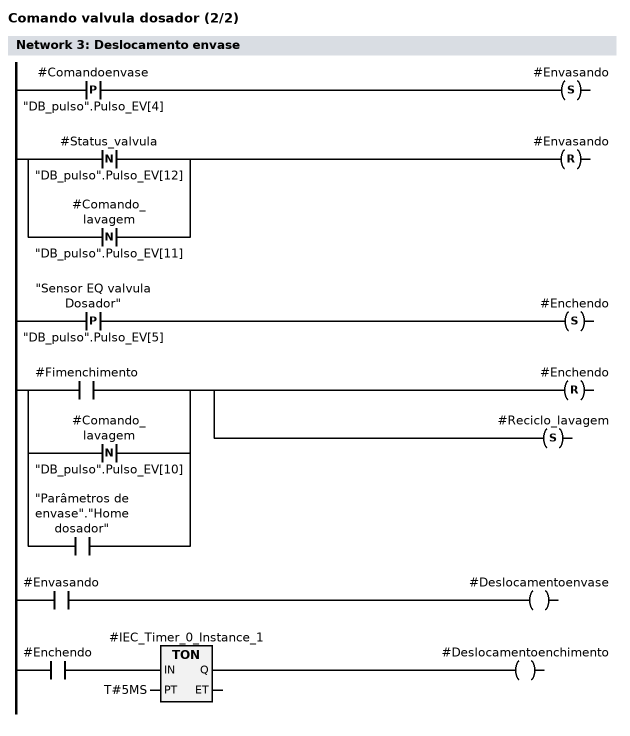
   #_w1 := #Comandoenvase AND NOT "DB_pulso".Pulso_EV[4];   // rising edge of #Comandoenvase
   "DB_pulso".Pulso_EV[4] := #Comandoenvase;
   IF #_w1 THEN #Envasando := TRUE; END_IF;
   #_w2 := NOT #Status_valvula AND "DB_pulso".Pulso_EV[12];   // falling edge of #Status_valvula
   "DB_pulso".Pulso_EV[12] := #Status_valvula;
   #_w3 := NOT #Comando_lavagem AND "DB_pulso".Pulso_EV[11];   // falling edge of #Comando_lavagem
   "DB_pulso".Pulso_EV[11] := #Comando_lavagem;
   IF #_w2 OR #_w3 THEN #Envasando := FALSE; END_IF;
   #_w4 := "Sensor EQ valvula Dosador" AND NOT "DB_pulso".Pulso_EV[5];   // rising edge of "Sensor EQ valvula Dosador"
   "DB_pulso".Pulso_EV[5] := "Sensor EQ valvula Dosador";
   IF #_w4 THEN #Enchendo := TRUE; END_IF;
   #_w5 := NOT #Comando_lavagem AND "DB_pulso".Pulso_EV[10];   // falling edge of #Comando_lavagem
   "DB_pulso".Pulso_EV[10] := #Comando_lavagem;
   IF #Fimenchimento OR #_w5 OR "Parâmetros de envase"."Home dosador" THEN
       #Enchendo := FALSE;
       #Reciclo_lavagem := TRUE;
   END_IF;
   #Deslocamentoenvase := #Envasando;
   #IEC_Timer_0_Instance_1(IN := #Enchendo, PT := T#5MS);   // TON
   #Deslocamentoenchimento := #IEC_Timer_0_Instance_1.Q;
END_REGION
END_FUNCTION_BLOCK

FUNCTION_BLOCK "Controle manipulador"   // FB4, LAD
{ S7_Optimized_Access := 'TRUE' }
VERSION : 0.1
   VAR_INPUT
      "Habilita comando" : Bool;
      "Pulso de movimento" : Bool;
      "Pulso pega tampa" : Bool;
      "Sensor cinlindro" : Bool;
      "Status Home" : Bool;
      Status_deslocamentoavanço : Bool;
      Status_deslocamentorecuo : Bool;
      Alvoa_atingidoavanço : Bool;
      Alvo_atingidorecuo : Bool;
      Fimenvase : Bool;
   END_VAR
   VAR_OUTPUT
      "Pulso avaço" : Bool;
      "Pulso recuo" : Bool;
      "Pulso posi_direito" : Bool;
      "Pulso posi_esquerdo" : Bool;
      "Cilindro manipulador" : Bool;
      "Cilindro empurrador" : Bool;
      "Valvula vacuo_1" : Bool;
      "Valvula sopro_1" : Bool;
      "Valvula vacuo_2" : Bool;
      "Valvula sopro_2" : Bool;
   END_VAR
   VAR
      Comandorodar : Bool;
      Status_pegatampa : Bool;
      IEC_Timer_0_Instance : TON_TIME;
      IEC_Timer_0_Instance_1 : TOF_TIME;
      IEC_Timer_0_Instance_2 : TOF_TIME;
      IEC_Timer_0_Instance_3 : TON_TIME;
   END_VAR
   VAR_TEMP   // added for the SCL form of the ladder/FBD networks
      _w1 : Bool;
      _w2 : Bool;
      _w3 : Bool;
      _w4 : Bool;
      _w5 : Bool;
      _w6 : Bool;
      _w7 : Bool;
      _w8 : Bool;
      _w9 : Bool;
      _w10 : Bool;
      _w11 : Bool;
   END_VAR
BEGIN

REGION Network 1: Habilita comando de transmissão
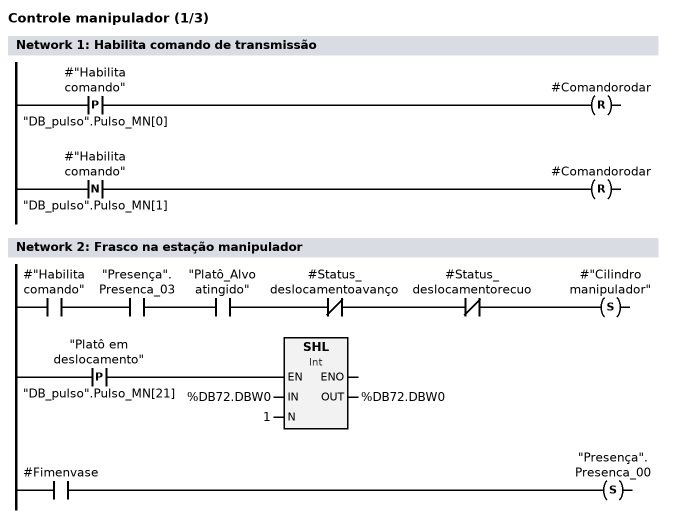
   RUNG wire#powerrail
      P_Contact(operand := #"Habilita comando", bit := "DB_pulso".Pulso_MN[0])
      R_Coil( #Comandorodar )
   END_RUNG
   RUNG wire#powerrail
      N_Contact(operand := #"Habilita comando", bit := "DB_pulso".Pulso_MN[1])
      R_Coil( #Comandorodar )
   END_RUNG
   // the same network as SCL:
   #_w1 := #"Habilita comando" AND NOT "DB_pulso".Pulso_MN[0];   // rising edge of #"Habilita comando"
   "DB_pulso".Pulso_MN[0] := #"Habilita comando";
   IF #_w1 THEN #Comandorodar := FALSE; END_IF;
   #_w2 := NOT #"Habilita comando" AND "DB_pulso".Pulso_MN[1];   // falling edge of #"Habilita comando"
   "DB_pulso".Pulso_MN[1] := #"Habilita comando";
   IF #_w2 THEN #Comandorodar := FALSE; END_IF;
END_REGION

REGION Network 2: Frasco na estação manipulador
   RUNG wire#powerrail
      Contact( #"Habilita comando" )
      Contact( "Presença".Presenca_03 )
      Contact( "Platô_Alvo atingido" )
      I_Contact( #Status_deslocamentoavanço )
      I_Contact( #Status_deslocamentorecuo )
      S_Coil( #"Cilindro manipulador" )
   END_RUNG
   RUNG wire#powerrail
      P_Contact(operand := "Platô em deslocamento", bit := "DB_pulso".Pulso_MN[21])
      { S7_Templates := "SrcType := Int" } Shl(in := %DB72.DBW0, n := 1, out => %DB72.DBW0)
   END_RUNG
   RUNG wire#powerrail
      Contact( #Fimenvase )
      S_Coil( "Presença".Presenca_00 )
   END_RUNG
   // the same network as SCL:
   IF #"Habilita comando" AND "Presença".Presenca_03 AND "Platô_Alvo atingido" AND NOT #Status_deslocamentoavanço AND NOT #Status_deslocamentorecuo THEN
       #"Cilindro manipulador" := TRUE;
   END_IF;
   #_w1 := "Platô em deslocamento" AND NOT "DB_pulso".Pulso_MN[21];   // rising edge of "Platô em deslocamento"
   "DB_pulso".Pulso_MN[21] := "Platô em deslocamento";
   IF #_w1 THEN %DB72.DBW0 := SHL(IN := %DB72.DBW0, N := 1); END_IF;
   IF #Fimenvase THEN "Presença".Presenca_00 := TRUE; END_IF;
END_REGION

REGION Network 3: Controle manipulador de tampa
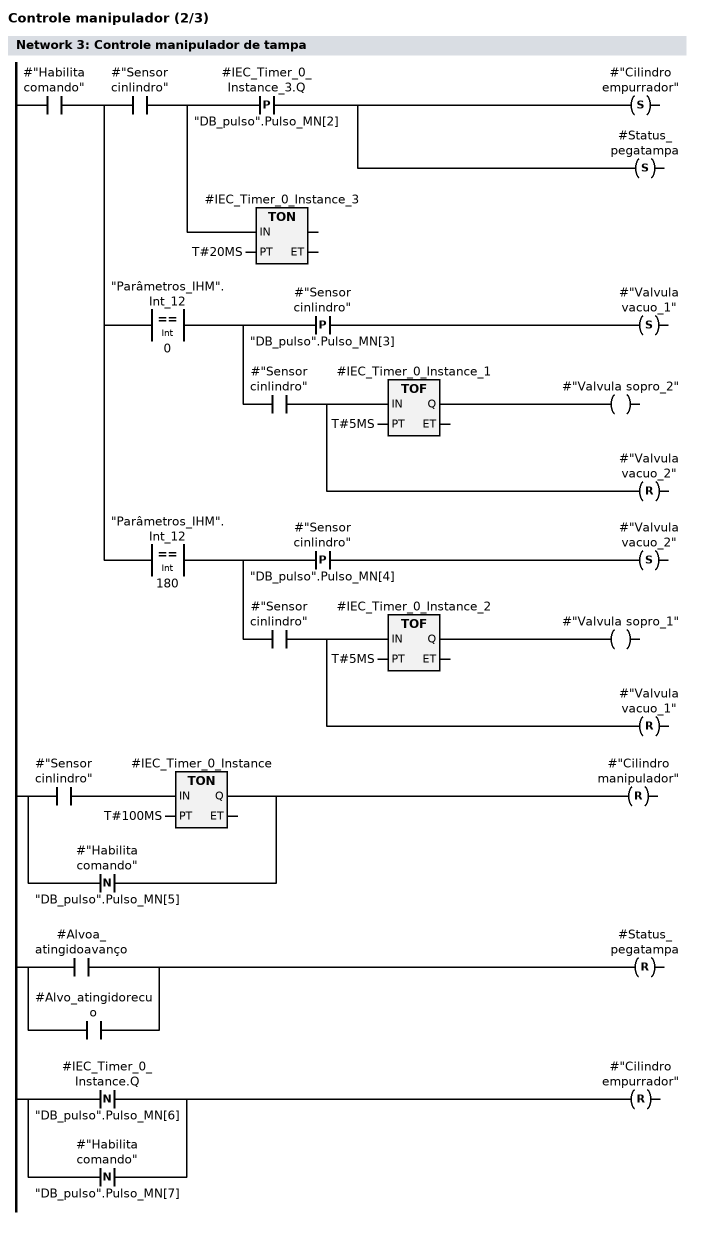
   #_w1 := #"Habilita comando" AND #"Sensor cinlindro";
   #_w2 := #_w1 AND #IEC_Timer_0_Instance_3.Q AND NOT "DB_pulso".Pulso_MN[2];   // rising edge of #IEC_Timer_0_Instance_3.Q
   "DB_pulso".Pulso_MN[2] := #IEC_Timer_0_Instance_3.Q;
   IF #_w2 THEN
       #"Cilindro empurrador" := TRUE;
       #Status_pegatampa := TRUE;
   END_IF;
   #IEC_Timer_0_Instance_3(IN := #_w1, PT := T#20MS);   // TON
   #_w3 := #"Habilita comando" AND ("Parâmetros_IHM".Int_12 = 0);
   #_w4 := #_w3 AND #"Sensor cinlindro" AND NOT "DB_pulso".Pulso_MN[3];   // rising edge of #"Sensor cinlindro"
   "DB_pulso".Pulso_MN[3] := #"Sensor cinlindro";
   IF #_w4 THEN #"Valvula vacuo_1" := TRUE; END_IF;
   #_w5 := #_w3 AND #"Sensor cinlindro";
   #IEC_Timer_0_Instance_1(IN := #_w5, PT := T#5MS);   // TOF
   #"Valvula sopro_2" := #IEC_Timer_0_Instance_1.Q;
   IF #_w5 THEN #"Valvula vacuo_2" := FALSE; END_IF;
   #_w6 := #"Habilita comando" AND ("Parâmetros_IHM".Int_12 = 180);
   #_w7 := #_w6 AND #"Sensor cinlindro" AND NOT "DB_pulso".Pulso_MN[4];   // rising edge of #"Sensor cinlindro"
   "DB_pulso".Pulso_MN[4] := #"Sensor cinlindro";
   IF #_w7 THEN #"Valvula vacuo_2" := TRUE; END_IF;
   #_w8 := #_w6 AND #"Sensor cinlindro";
   #IEC_Timer_0_Instance_2(IN := #_w8, PT := T#5MS);   // TOF
   #"Valvula sopro_1" := #IEC_Timer_0_Instance_2.Q;
   IF #_w8 THEN #"Valvula vacuo_1" := FALSE; END_IF;
   #IEC_Timer_0_Instance(IN := #"Sensor cinlindro", PT := T#100MS);   // TON
   #_w9 := NOT #"Habilita comando" AND "DB_pulso".Pulso_MN[5];   // falling edge of #"Habilita comando"
   "DB_pulso".Pulso_MN[5] := #"Habilita comando";
   IF #IEC_Timer_0_Instance.Q OR #_w9 THEN #"Cilindro manipulador" := FALSE; END_IF;
   IF #Alvoa_atingidoavanço OR #Alvo_atingidorecuo THEN #Status_pegatampa := FALSE; END_IF;
   #_w10 := NOT #IEC_Timer_0_Instance.Q AND "DB_pulso".Pulso_MN[6];   // falling edge of #IEC_Timer_0_Instance.Q
   "DB_pulso".Pulso_MN[6] := #IEC_Timer_0_Instance.Q;
   #_w11 := NOT #"Habilita comando" AND "DB_pulso".Pulso_MN[7];   // falling edge of #"Habilita comando"
   "DB_pulso".Pulso_MN[7] := #"Habilita comando";
   IF #_w10 OR #_w11 THEN #"Cilindro empurrador" := FALSE; END_IF;
END_REGION

REGION Network 4: Controle deslocamento manipulador
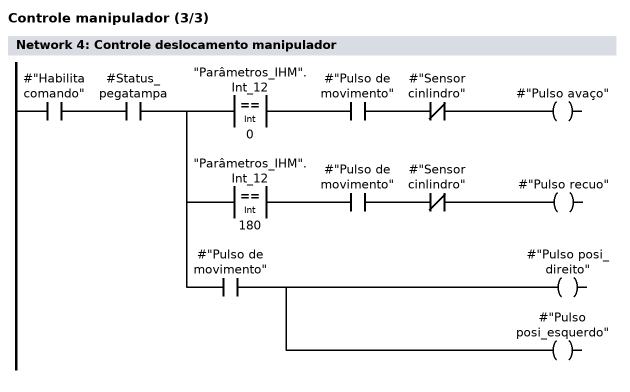
   RUNG wire#powerrail
      Contact( #"Habilita comando" )
      Contact( #Status_pegatampa )
      wire#w1
      { S7_Templates := "SrcType := Int" } EQ_Contact(in1 := "Parâmetros_IHM".Int_12, in2 := 0)
      Contact( #"Pulso de movimento" )
      I_Contact( #"Sensor cinlindro" )
      Coil( #"Pulso avaço" )
   END_RUNG
   RUNG wire#w1
      { S7_Templates := "SrcType := Int" } EQ_Contact(in1 := "Parâmetros_IHM".Int_12, in2 := 180)
      Contact( #"Pulso de movimento" )
      I_Contact( #"Sensor cinlindro" )
      Coil( #"Pulso recuo" )
   END_RUNG
   RUNG wire#w1
      Contact( #"Pulso de movimento" )
      wire#w2
      Coil( #"Pulso posi_direito" )
   END_RUNG
   RUNG wire#w2
      Coil( #"Pulso posi_esquerdo" )
   END_RUNG
   // the same network as SCL:
   #_w1 := #"Habilita comando" AND #Status_pegatampa;
   #"Pulso avaço" := #_w1 AND ("Parâmetros_IHM".Int_12 = 0) AND #"Pulso de movimento" AND NOT #"Sensor cinlindro";
   #"Pulso recuo" := #_w1 AND ("Parâmetros_IHM".Int_12 = 180) AND #"Pulso de movimento" AND NOT #"Sensor cinlindro";
   #"Pulso posi_direito" := #_w1 AND #"Pulso de movimento";
   #"Pulso posi_esquerdo" := #"Pulso posi_direito";
END_REGION
END_FUNCTION_BLOCK

FUNCTION_BLOCK "Rosqueador_tampa"   // FB5, LAD
{ S7_Optimized_Access := 'TRUE' }
VERSION : 0.1
   VAR_INPUT
      Habilita_comando : Bool;
      Sensor_tamap : Bool;
      Sensor_Cilindro : Bool;
      Desce_rosqueador : Bool;
      Continuo : Bool;
      Manual_decse : Bool;
      Manual_ciclo : Bool;
      Alvo_atingido : Bool;
      Timer_Rosqueador : Time;
      Timer_inicio_fechamento : Time;
   END_VAR
   VAR_OUTPUT
      Cilindro : Bool;
      Rosqueador_pulso : Bool;
      Rosqueador_Jog : Bool;
      Rosqueador_emdeslocamento : Bool;
      Timer_real : Time;
   END_VAR
   VAR
      Comando_ON : Bool;
      Status_Cilindro : Bool;
      Presença_tampa : Bool;
      IEC_Timer_0_Instance : TON_TIME;
      IEC_Timer_0_Instance_1 : TON_TIME;
   END_VAR
   VAR_TEMP   // added for the SCL form of the ladder/FBD networks
      _w1 : Bool;
      _w2 : Bool;
      _w3 : Bool;
      _w4 : Bool;
      _w5 : Bool;
      _w6 : Bool;
   END_VAR
BEGIN

REGION Network 1: Habilita Comando
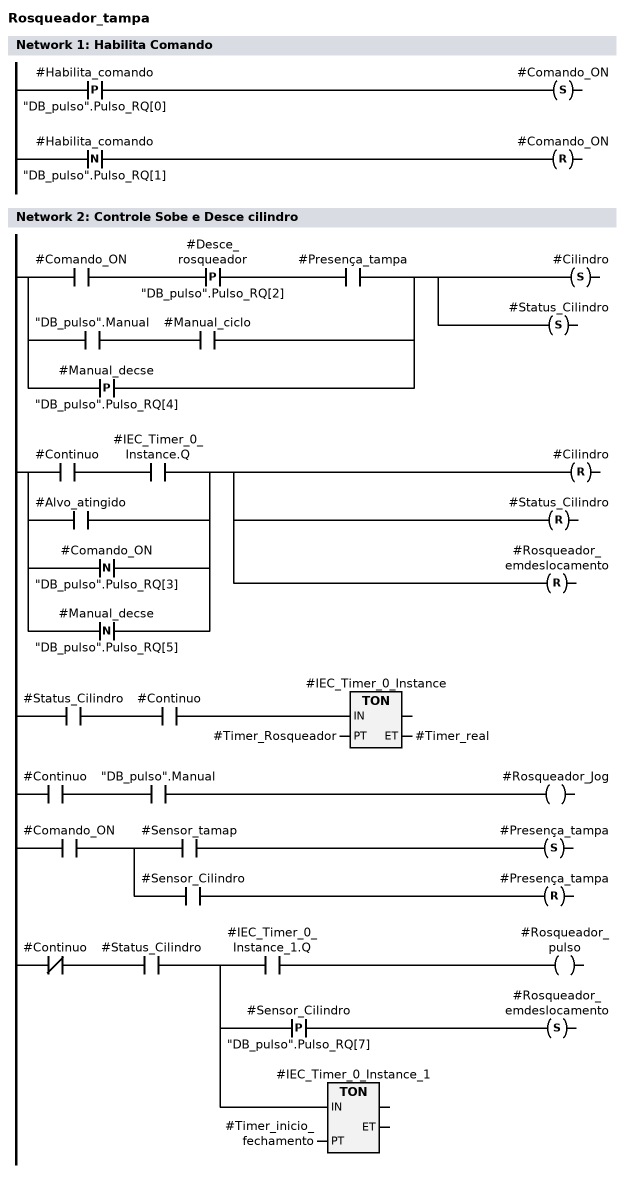
   RUNG wire#powerrail
      P_Contact(operand := #Habilita_comando, bit := "DB_pulso".Pulso_RQ[0])
      S_Coil( #Comando_ON )
   END_RUNG
   RUNG wire#powerrail
      N_Contact(operand := #Habilita_comando, bit := "DB_pulso".Pulso_RQ[1])
      R_Coil( #Comando_ON )
   END_RUNG
   // the same network as SCL:
   #_w1 := #Habilita_comando AND NOT "DB_pulso".Pulso_RQ[0];   // rising edge of #Habilita_comando
   "DB_pulso".Pulso_RQ[0] := #Habilita_comando;
   IF #_w1 THEN #Comando_ON := TRUE; END_IF;
   #_w2 := NOT #Habilita_comando AND "DB_pulso".Pulso_RQ[1];   // falling edge of #Habilita_comando
   "DB_pulso".Pulso_RQ[1] := #Habilita_comando;
   IF #_w2 THEN #Comando_ON := FALSE; END_IF;
END_REGION

REGION Network 2: Controle Sobe e Desce cilindro
   #_w1 := #Comando_ON AND #Desce_rosqueador AND NOT "DB_pulso".Pulso_RQ[2];   // rising edge of #Desce_rosqueador
   "DB_pulso".Pulso_RQ[2] := #Desce_rosqueador;
   #_w2 := #Manual_decse AND NOT "DB_pulso".Pulso_RQ[4];   // rising edge of #Manual_decse
   "DB_pulso".Pulso_RQ[4] := #Manual_decse;
   IF (#_w1 AND #Presença_tampa) OR ("DB_pulso".Manual AND #Manual_ciclo) OR #_w2 THEN
       #Cilindro := TRUE;
       #Status_Cilindro := TRUE;
   END_IF;
   #_w3 := NOT #Comando_ON AND "DB_pulso".Pulso_RQ[3];   // falling edge of #Comando_ON
   "DB_pulso".Pulso_RQ[3] := #Comando_ON;
   #_w4 := NOT #Manual_decse AND "DB_pulso".Pulso_RQ[5];   // falling edge of #Manual_decse
   "DB_pulso".Pulso_RQ[5] := #Manual_decse;
   IF (#Continuo AND #IEC_Timer_0_Instance.Q) OR #Alvo_atingido OR #_w3 OR #_w4 THEN
       #Cilindro := FALSE;
       #Status_Cilindro := FALSE;
       #Rosqueador_emdeslocamento := FALSE;
   END_IF;
   #IEC_Timer_0_Instance(IN := #Status_Cilindro AND #Continuo, PT := #Timer_Rosqueador, ET => #Timer_real);   // TON
   #Rosqueador_Jog := #Continuo AND "DB_pulso".Manual;
   IF #Comando_ON AND #Sensor_tamap THEN #Presença_tampa := TRUE; END_IF;
   IF #Comando_ON AND #Sensor_Cilindro THEN #Presença_tampa := FALSE; END_IF;
   #_w5 := NOT #Continuo AND #Status_Cilindro;
   #Rosqueador_pulso := #_w5 AND #IEC_Timer_0_Instance_1.Q;
   #_w6 := #_w5 AND #Sensor_Cilindro AND NOT "DB_pulso".Pulso_RQ[7];   // rising edge of #Sensor_Cilindro
   "DB_pulso".Pulso_RQ[7] := #Sensor_Cilindro;
   IF #_w6 THEN #Rosqueador_emdeslocamento := TRUE; END_IF;
   #IEC_Timer_0_Instance_1(IN := #_w5, PT := #Timer_inicio_fechamento);   // TON
END_REGION
END_FUNCTION_BLOCK

FUNCTION "Transmissão Estrela" : Void   // FC1, LAD
{ S7_Optimized_Access := 'TRUE' }
VERSION : 0.1
   VAR_INPUT
      "IN deslocamento" : Bool;
   END_VAR
   VAR_TEMP   // added for the SCL form of the ladder/FBD networks
      _w1 : Bool;
   END_VAR
BEGIN

REGION Network 1: Habilita servo drive estrela
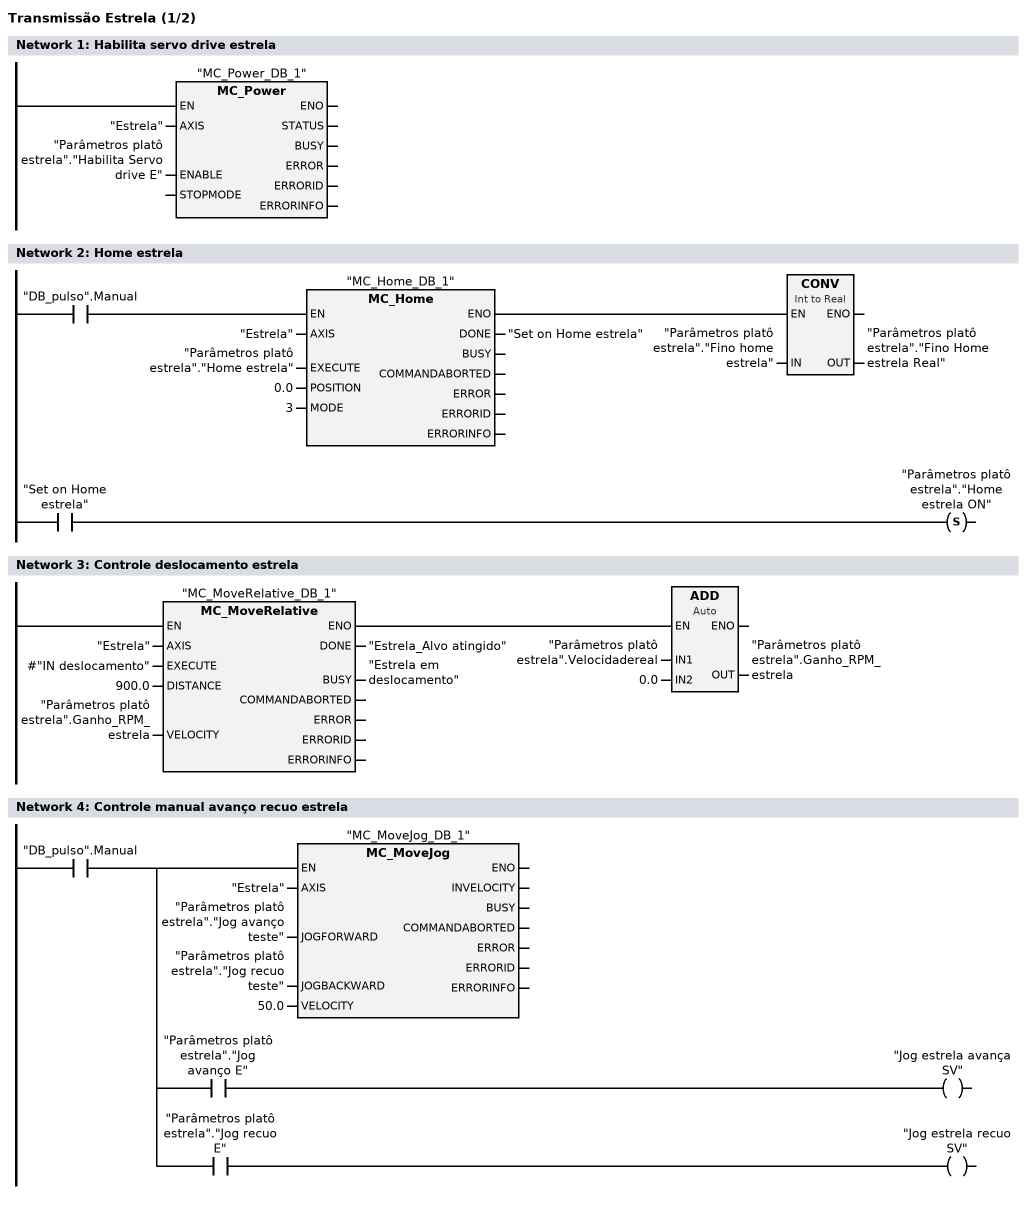
   "MC_Power_DB_1"(Axis := "Estrela", Enable := "Parâmetros platô estrela"."Habilita Servo drive E");   // MC_Power
END_REGION

REGION Network 2: Home estrela
   // ENO of a box is taken as its EN; it also drops when the box reports an error
   #_w1 := "DB_pulso".Manual;
   IF #_w1 THEN
       "MC_Home_DB_1"(Axis := "Estrela",   // MC_Home
                      Execute := "Parâmetros platô estrela"."Home estrela",
                      Position := 0.0,
                      Mode := 3,
                      Done => "Set on Home estrela");
       "Parâmetros platô estrela"."Fino Home estrela Real" := INT_TO_REAL("Parâmetros platô estrela"."Fino home estrela");
   END_IF;
   IF "Set on Home estrela" THEN "Parâmetros platô estrela"."Home estrela ON" := TRUE; END_IF;
END_REGION

REGION Network 3: Controle deslocamento estrela
   // ENO of a box is taken as its EN; it also drops when the box reports an error
   "MC_MoveRelative_DB_1"(Axis := "Estrela",   // MC_MoveRelative
                          Execute := #"IN deslocamento",
                          Distance := 900.0,
                          Velocity := "Parâmetros platô estrela".Ganho_RPM_estrela,
                          Done => "Estrela_Alvo atingido",
                          Busy => "Estrela em deslocamento");
   "Parâmetros platô estrela".Ganho_RPM_estrela := "Parâmetros platô estrela".Velocidadereal + 0.0;
END_REGION

REGION Network 4: Controle manual avanço recuo estrela
   #_w1 := "DB_pulso".Manual;
   IF #_w1 THEN
       "MC_MoveJog_DB_1"(Axis := "Estrela",   // MC_MoveJog
                         JogForward := "Parâmetros platô estrela"."Jog avanço teste",
                         JogBackward := "Parâmetros platô estrela"."Jog recuo teste",
                         Velocity := 50.0);
   END_IF;
   "Jog estrela avança SV" := #_w1 AND "Parâmetros platô estrela"."Jog avanço E";
   "Jog estrela recuo SV" := #_w1 AND "Parâmetros platô estrela"."Jog recuo E";
END_REGION

REGION Network 5: Controle de rampa de aceseleração e desaceleração
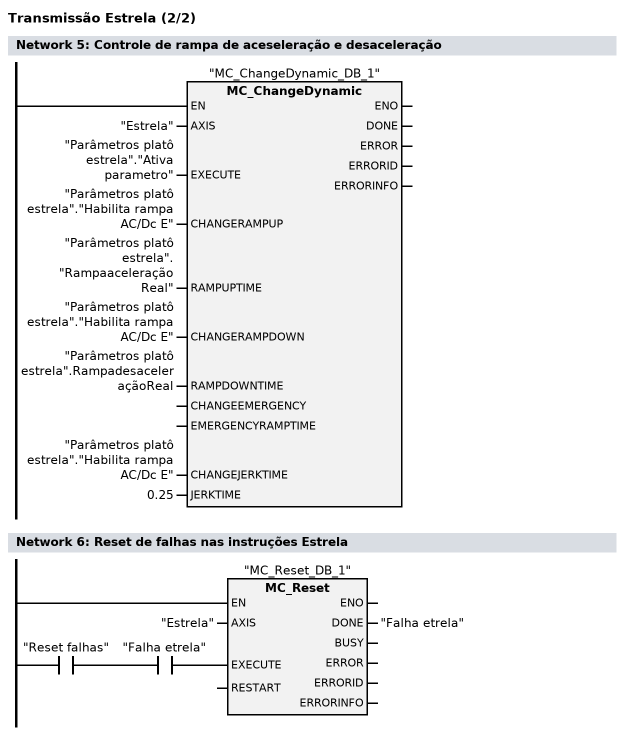
   "MC_ChangeDynamic_DB_1"(Axis := "Estrela",   // MC_ChangeDynamic
                           Execute := "Parâmetros platô estrela"."Ativa parametro",
                           ChangeRampUp := "Parâmetros platô estrela"."Habilita rampa AC/Dc E",
                           RampUpTime := "Parâmetros platô estrela"."Rampaaceleração Real",
                           ChangeRampDown := "Parâmetros platô estrela"."Habilita rampa AC/Dc E",
                           RampDownTime := "Parâmetros platô estrela".RampadesaceleraçãoReal,
                           ChangeJerkTime := "Parâmetros platô estrela"."Habilita rampa AC/Dc E",
                           JerkTime := 0.25);
END_REGION

REGION Network 6: Reset de falhas nas instruções Estrela
   "MC_Reset_DB_1"(Axis := "Estrela", Execute := "Reset falhas" AND "Falha etrela", Done => "Falha etrela");   // MC_Reset
END_REGION
END_FUNCTION

FUNCTION "Transmissão Platô" : Void   // FC2, LAD
{ S7_Optimized_Access := 'TRUE' }
VERSION : 0.1
   VAR_INPUT
      "IN deslocamento" : Bool;
   END_VAR
   VAR_TEMP   // added for the SCL form of the ladder/FBD networks
      _w1 : Bool;
   END_VAR
BEGIN

REGION Network 1: Habilita servo drive platô
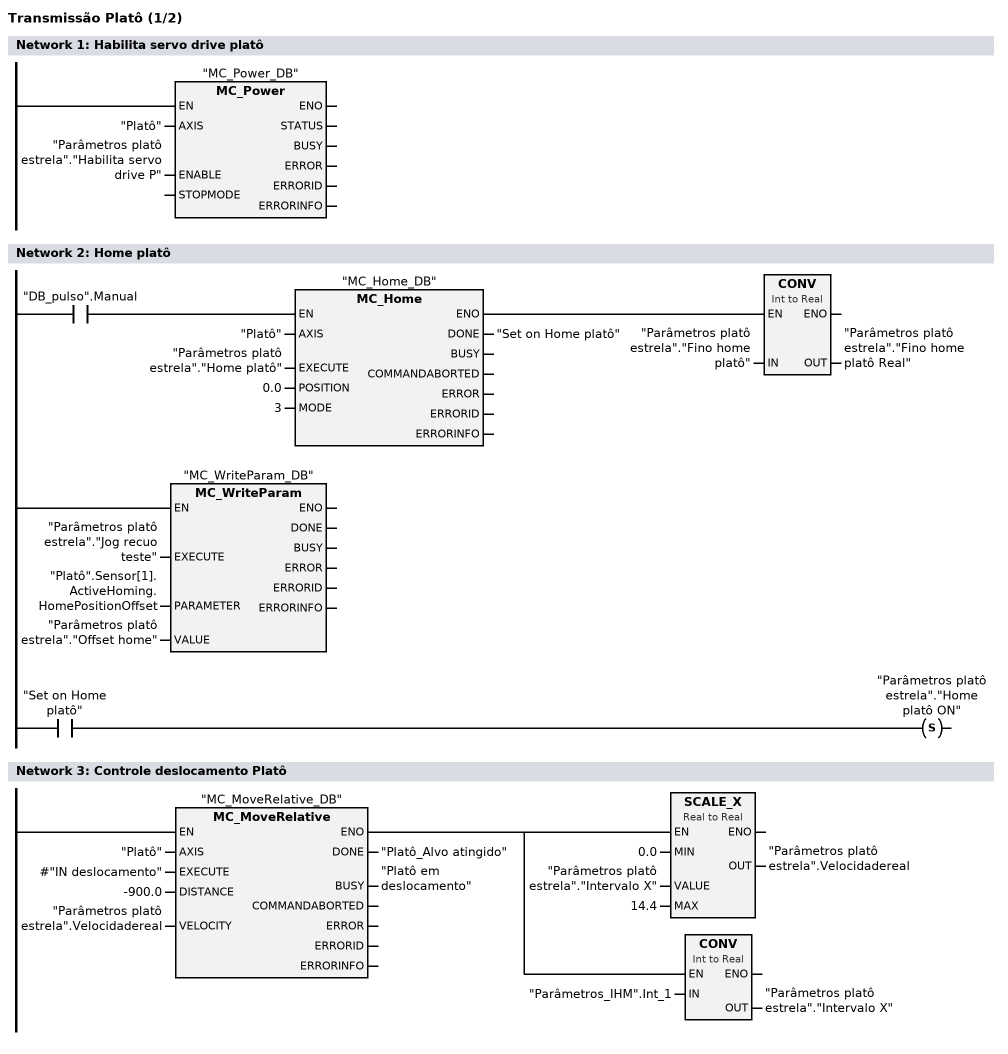
   "MC_Power_DB"(Axis := "Platô", Enable := "Parâmetros platô estrela"."Habilita servo drive P");   // MC_Power
END_REGION

REGION Network 2: Home platô
   // ENO of a box is taken as its EN; it also drops when the box reports an error
   #_w1 := "DB_pulso".Manual;
   IF #_w1 THEN
       "MC_Home_DB"(Axis := "Platô",   // MC_Home
                    Execute := "Parâmetros platô estrela"."Home platô",
                    Position := 0.0,
                    Mode := 3,
                    Done => "Set on Home platô");
       "Parâmetros platô estrela"."Fino home platô Real" := INT_TO_REAL("Parâmetros platô estrela"."Fino home platô");
   END_IF;
   "MC_WriteParam_DB"(Execute := "Parâmetros platô estrela"."Jog recuo teste",   // MC_WriteParam
                      Parameter := "Platô".Sensor[1].ActiveHoming.HomePositionOffset,
                      Value := "Parâmetros platô estrela"."Offset home");
   IF "Set on Home platô" THEN "Parâmetros platô estrela"."Home platô ON" := TRUE; END_IF;
END_REGION

REGION Network 3: Controle deslocamento Platô
   // ENO of a box is taken as its EN; it also drops when the box reports an error
   "MC_MoveRelative_DB"(Axis := "Platô",   // MC_MoveRelative
                        Execute := #"IN deslocamento",
                        Distance := -900.0,
                        Velocity := "Parâmetros platô estrela".Velocidadereal,
                        Done => "Platô_Alvo atingido",
                        Busy => "Platô em deslocamento");
   "Parâmetros platô estrela".Velocidadereal := SCALE_X(MIN := 0.0, VALUE := "Parâmetros platô estrela"."Intervalo X", MAX := 14.4);
   "Parâmetros platô estrela"."Intervalo X" := INT_TO_REAL("Parâmetros_IHM".Int_1);
END_REGION

REGION Network 4: Controle Manual avança reucuo transmissão platô estrela
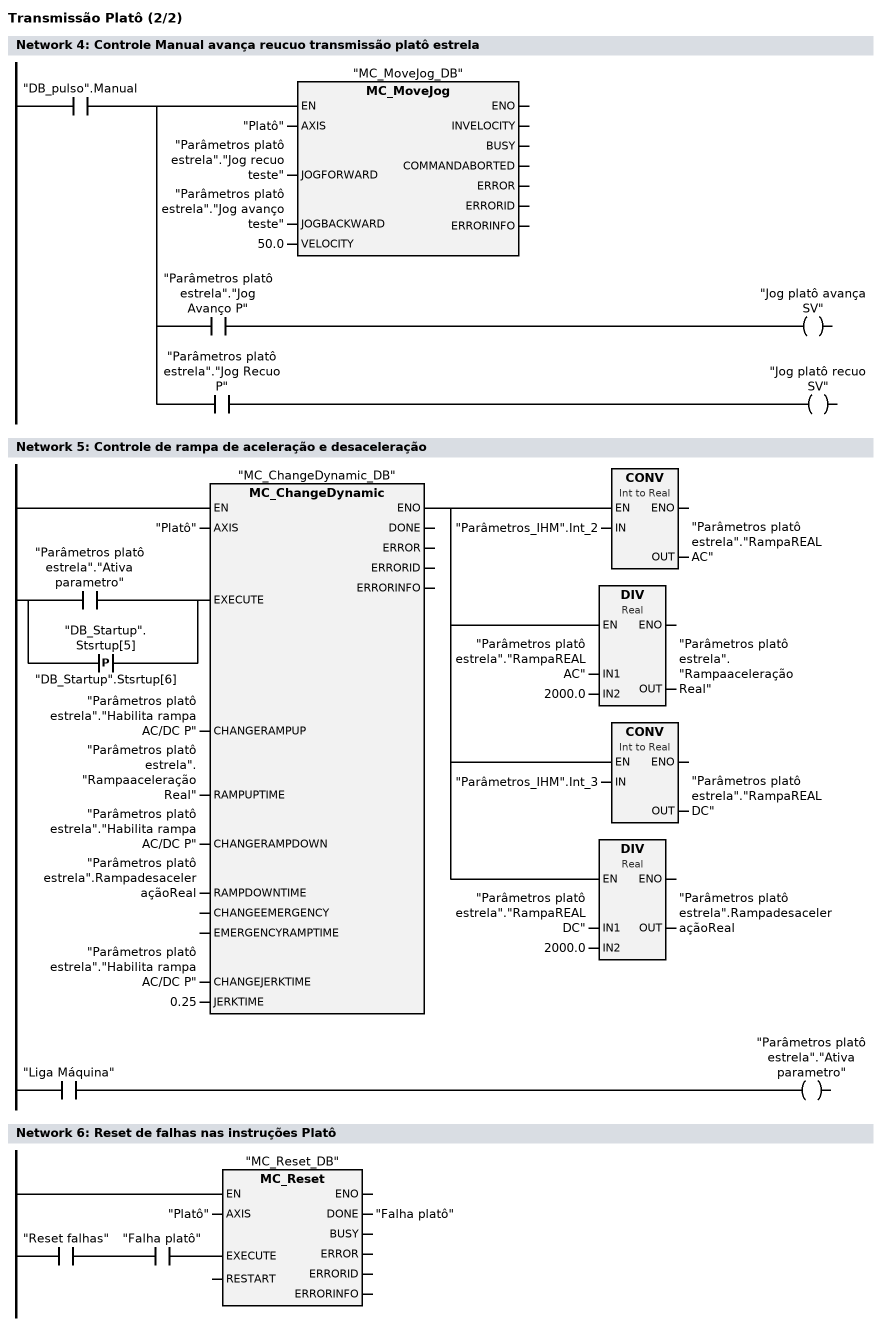
   #_w1 := "DB_pulso".Manual;
   IF #_w1 THEN
       "MC_MoveJog_DB"(Axis := "Platô",   // MC_MoveJog
                       JogForward := "Parâmetros platô estrela"."Jog recuo teste",
                       JogBackward := "Parâmetros platô estrela"."Jog avanço teste",
                       Velocity := 50.0);
   END_IF;
   "Jog platô avança SV" := #_w1 AND "Parâmetros platô estrela"."Jog Avanço P";
   "Jog platô recuo SV" := #_w1 AND "Parâmetros platô estrela"."Jog Recuo P";
END_REGION

REGION Network 5: Controle de rampa de aceleração e desaceleração
   // ENO of a box is taken as its EN; it also drops when the box reports an error
   #_w1 := "DB_Startup".Stsrtup[5] AND NOT "DB_Startup".Stsrtup[6];   // rising edge of "DB_Startup".Stsrtup[5]
   "DB_Startup".Stsrtup[6] := "DB_Startup".Stsrtup[5];
   "MC_ChangeDynamic_DB"(Axis := "Platô",   // MC_ChangeDynamic
                         Execute := "Parâmetros platô estrela"."Ativa parametro" OR #_w1,
                         ChangeRampUp := "Parâmetros platô estrela"."Habilita rampa AC/DC P",
                         RampUpTime := "Parâmetros platô estrela"."Rampaaceleração Real",
                         ChangeRampDown := "Parâmetros platô estrela"."Habilita rampa AC/DC P",
                         RampDownTime := "Parâmetros platô estrela".RampadesaceleraçãoReal,
                         ChangeJerkTime := "Parâmetros platô estrela"."Habilita rampa AC/DC P",
                         JerkTime := 0.25);
   "Parâmetros platô estrela"."RampaREAL AC" := INT_TO_REAL("Parâmetros_IHM".Int_2);
   "Parâmetros platô estrela"."Rampaaceleração Real" := "Parâmetros platô estrela"."RampaREAL AC" / 2000.0;
   "Parâmetros platô estrela"."RampaREAL DC" := INT_TO_REAL("Parâmetros_IHM".Int_3);
   "Parâmetros platô estrela".RampadesaceleraçãoReal := "Parâmetros platô estrela"."RampaREAL DC" / 2000.0;
   "Parâmetros platô estrela"."Ativa parametro" := "Liga Máquina";
END_REGION

REGION Network 6: Reset de falhas nas instruções Platô
   "MC_Reset_DB"(Axis := "Platô", Execute := "Reset falhas" AND "Falha platô", Done => "Falha platô");   // MC_Reset
END_REGION
END_FUNCTION

FUNCTION "Controle envase" : Void   // FC3, LAD
{ S7_Optimized_Access := 'TRUE' }
VERSION : 0.1
   VAR_INPUT
      Envasar : Bool;
      Enchimento : Bool;
   END_VAR
   VAR_TEMP   // added for the SCL form of the ladder/FBD networks
      _w1 : Bool;
   END_VAR
BEGIN

REGION Network 1: Habilita servo drive envase
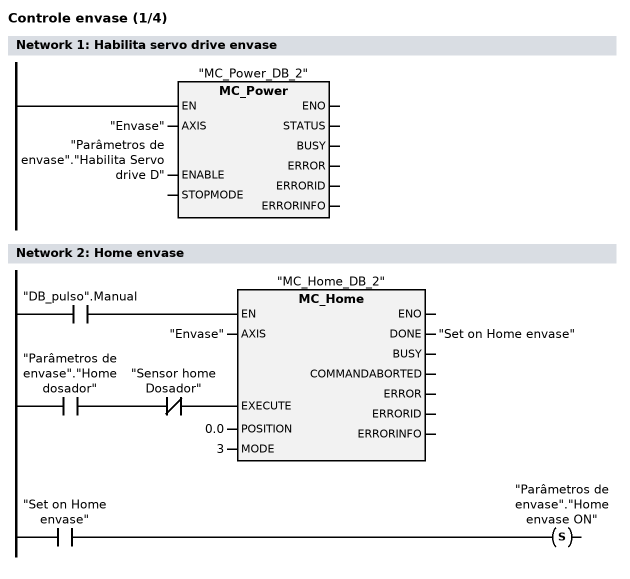
   "MC_Power_DB_2"(Axis := "Envase", Enable := "Parâmetros de envase"."Habilita Servo drive D");   // MC_Power
END_REGION

REGION Network 2: Home envase
   IF "DB_pulso".Manual THEN
       "MC_Home_DB_2"(Axis := "Envase",   // MC_Home
                      Execute := "Parâmetros de envase"."Home dosador" AND NOT "Sensor home Dosador",
                      Position := 0.0,
                      Mode := 3,
                      Done => "Set on Home envase");
   END_IF;
   IF "Set on Home envase" THEN "Parâmetros de envase"."Home envase ON" := TRUE; END_IF;
END_REGION

REGION Network 3: Controle deslocamento envase
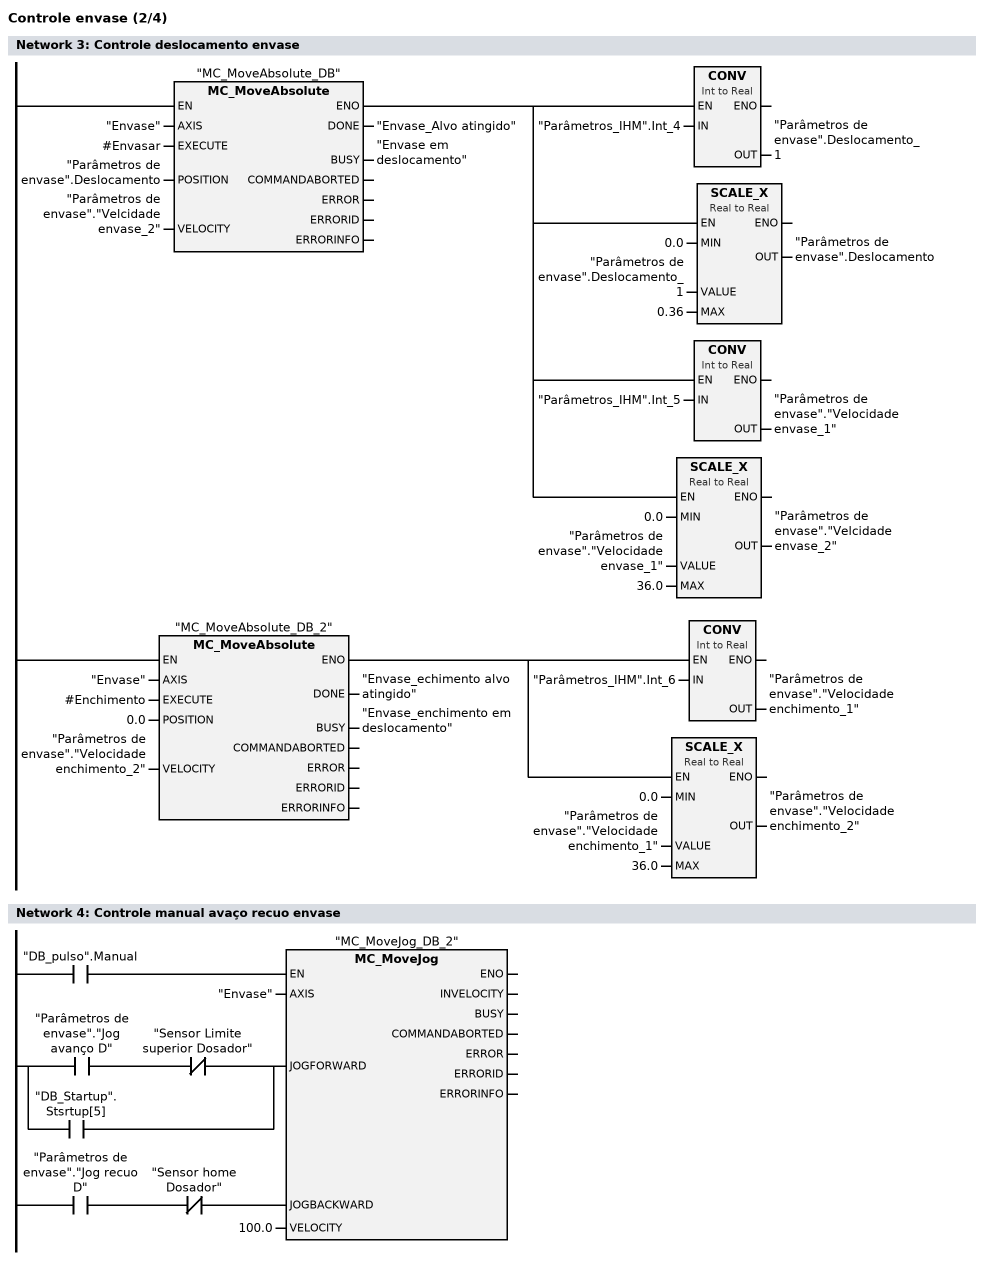
   // ENO of a box is taken as its EN; it also drops when the box reports an error
   "MC_MoveAbsolute_DB"(Axis := "Envase",   // MC_MoveAbsolute
                        Execute := #Envasar,
                        Position := "Parâmetros de envase".Deslocamento,
                        Velocity := "Parâmetros de envase"."Velcidade envase_2",
                        Done => "Envase_Alvo atingido",
                        Busy => "Envase em deslocamento");
   "Parâmetros de envase".Deslocamento_1 := INT_TO_REAL("Parâmetros_IHM".Int_4);
   "Parâmetros de envase".Deslocamento := SCALE_X(MIN := 0.0, VALUE := "Parâmetros de envase".Deslocamento_1, MAX := 0.36);
   "Parâmetros de envase"."Velocidade envase_1" := INT_TO_REAL("Parâmetros_IHM".Int_5);
   "Parâmetros de envase"."Velcidade envase_2" := SCALE_X(MIN := 0.0, VALUE := "Parâmetros de envase"."Velocidade envase_1", MAX := 36.0);
   "MC_MoveAbsolute_DB_2"(Axis := "Envase",   // MC_MoveAbsolute
                          Execute := #Enchimento,
                          Position := 0.0,
                          Velocity := "Parâmetros de envase"."Velocidade enchimento_2",
                          Done => "Envase_echimento alvo atingido",
                          Busy => "Envase_enchimento em deslocamento");
   "Parâmetros de envase"."Velocidade enchimento_1" := INT_TO_REAL("Parâmetros_IHM".Int_6);
   "Parâmetros de envase"."Velocidade enchimento_2" := SCALE_X(MIN := 0.0, VALUE := "Parâmetros de envase"."Velocidade enchimento_1", MAX := 36.0);
END_REGION

REGION Network 4: Controle manual avaço recuo envase
   IF "DB_pulso".Manual THEN
       "MC_MoveJog_DB_2"(Axis := "Envase",   // MC_MoveJog
                         JogForward := ("Parâmetros de envase"."Jog avanço D" AND NOT "Sensor Limite superior Dosador") OR "DB_Startup".Stsrtup[5],
                         JogBackward := "Parâmetros de envase"."Jog recuo D" AND NOT "Sensor home Dosador",
                         Velocity := 100.0);
   END_IF;
END_REGION

REGION Network 5: Startup
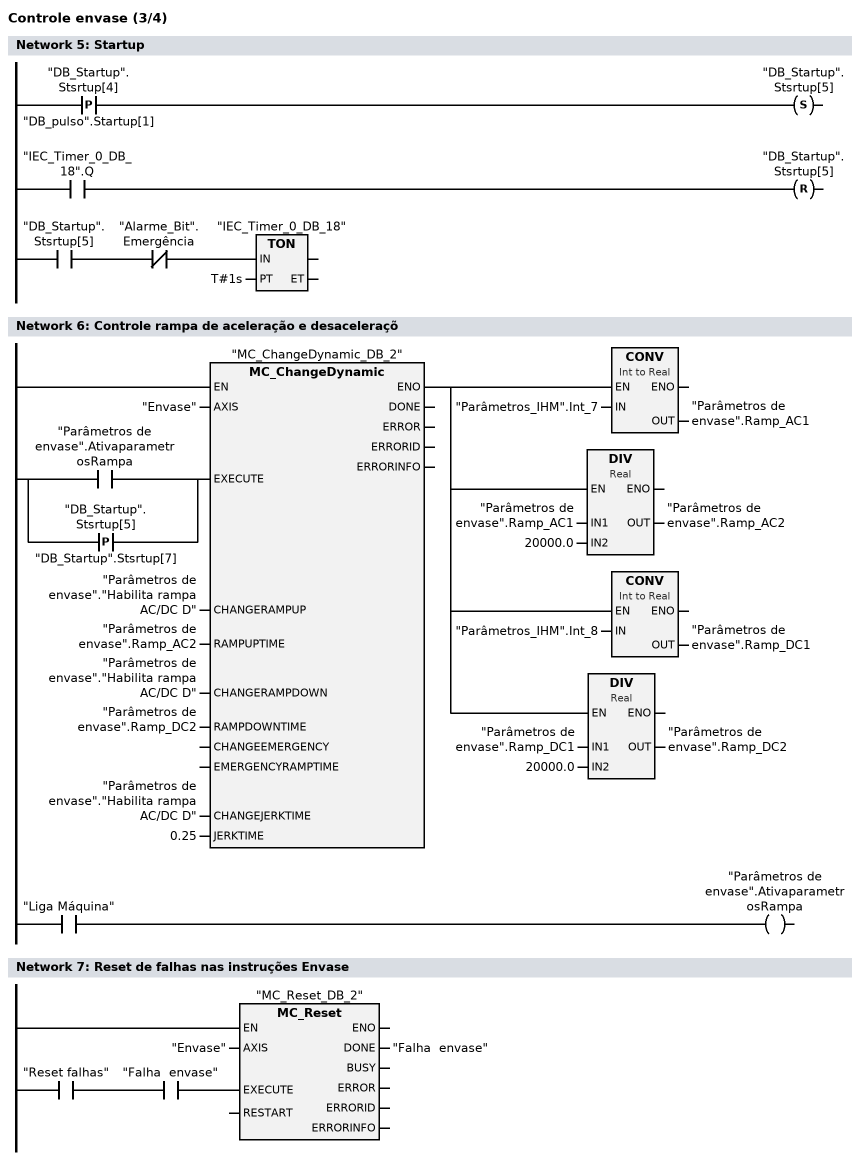
   #_w1 := "DB_Startup".Stsrtup[4] AND NOT "DB_pulso".Startup[1];   // rising edge of "DB_Startup".Stsrtup[4]
   "DB_pulso".Startup[1] := "DB_Startup".Stsrtup[4];
   IF #_w1 THEN "DB_Startup".Stsrtup[5] := TRUE; END_IF;
   IF "IEC_Timer_0_DB_18".Q THEN "DB_Startup".Stsrtup[5] := FALSE; END_IF;
   "IEC_Timer_0_DB_18".TON(IN := "DB_Startup".Stsrtup[5] AND NOT "Alarme_Bit".Emergência, PT := T#1s);
END_REGION

REGION Network 6: Controle rampa de aceleração e desaceleraçõ
   // ENO of a box is taken as its EN; it also drops when the box reports an error
   #_w1 := "DB_Startup".Stsrtup[5] AND NOT "DB_Startup".Stsrtup[7];   // rising edge of "DB_Startup".Stsrtup[5]
   "DB_Startup".Stsrtup[7] := "DB_Startup".Stsrtup[5];
   "MC_ChangeDynamic_DB_2"(Axis := "Envase",   // MC_ChangeDynamic
                           Execute := "Parâmetros de envase".AtivaparametrosRampa OR #_w1,
                           ChangeRampUp := "Parâmetros de envase"."Habilita rampa AC/DC D",
                           RampUpTime := "Parâmetros de envase".Ramp_AC2,
                           ChangeRampDown := "Parâmetros de envase"."Habilita rampa AC/DC D",
                           RampDownTime := "Parâmetros de envase".Ramp_DC2,
                           ChangeJerkTime := "Parâmetros de envase"."Habilita rampa AC/DC D",
                           JerkTime := 0.25);
   "Parâmetros de envase".Ramp_AC1 := INT_TO_REAL("Parâmetros_IHM".Int_7);
   "Parâmetros de envase".Ramp_AC2 := "Parâmetros de envase".Ramp_AC1 / 20000.0;
   "Parâmetros de envase".Ramp_DC1 := INT_TO_REAL("Parâmetros_IHM".Int_8);
   "Parâmetros de envase".Ramp_DC2 := "Parâmetros de envase".Ramp_DC1 / 20000.0;
   "Parâmetros de envase".AtivaparametrosRampa := "Liga Máquina";
END_REGION

REGION Network 7: Reset de falhas nas instruções Envase
   "MC_Reset_DB_2"(Axis := "Envase", Execute := "Reset falhas" AND "Falha  envase", Done => "Falha  envase");   // MC_Reset
END_REGION

REGION Network 8: Leitura deslocamento
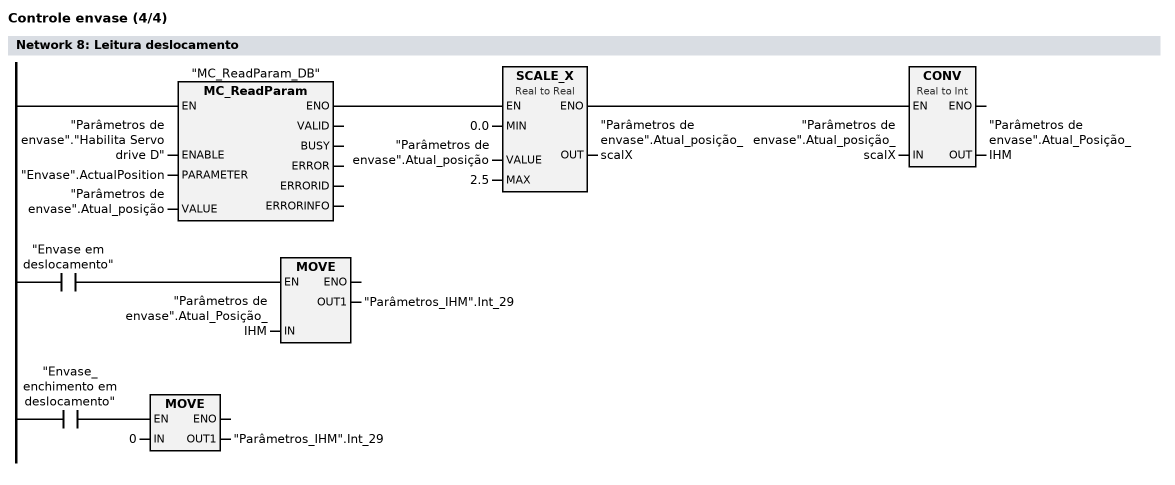
   // ENO of a box is taken as its EN; it also drops when the box reports an error
   "MC_ReadParam_DB"(Enable := "Parâmetros de envase"."Habilita Servo drive D",   // MC_ReadParam
                     Parameter := "Envase".ActualPosition,
                     Value := "Parâmetros de envase".Atual_posição);
   "Parâmetros de envase".Atual_posição_scalX := SCALE_X(MIN := 0.0, VALUE := "Parâmetros de envase".Atual_posição, MAX := 2.5);
   "Parâmetros de envase".Atual_Posição_IHM := REAL_TO_INT("Parâmetros de envase".Atual_posição_scalX);
   IF "Envase em deslocamento" THEN
       "Parâmetros_IHM".Int_29 := "Parâmetros de envase".Atual_Posição_IHM;
   END_IF;
   IF "Envase_enchimento em deslocamento" THEN "Parâmetros_IHM".Int_29 := 0; END_IF;
END_REGION
END_FUNCTION

FUNCTION "Manipulador" : Void   // FC4, LAD
{ S7_Optimized_Access := 'TRUE' }
VERSION : 0.1
   VAR_INPUT
      Avança : Bool;
      Recuo : Bool;
   END_VAR
   VAR_OUTPUT
      "Home posi direito" : Bool;
      "Home posi esquerdo" : Bool;
   END_VAR
   VAR_TEMP   // added for the SCL form of the ladder/FBD networks
      _w1 : Bool;
      _w2 : Bool;
   END_VAR
BEGIN

REGION Network 1: Habilita Drive STR8
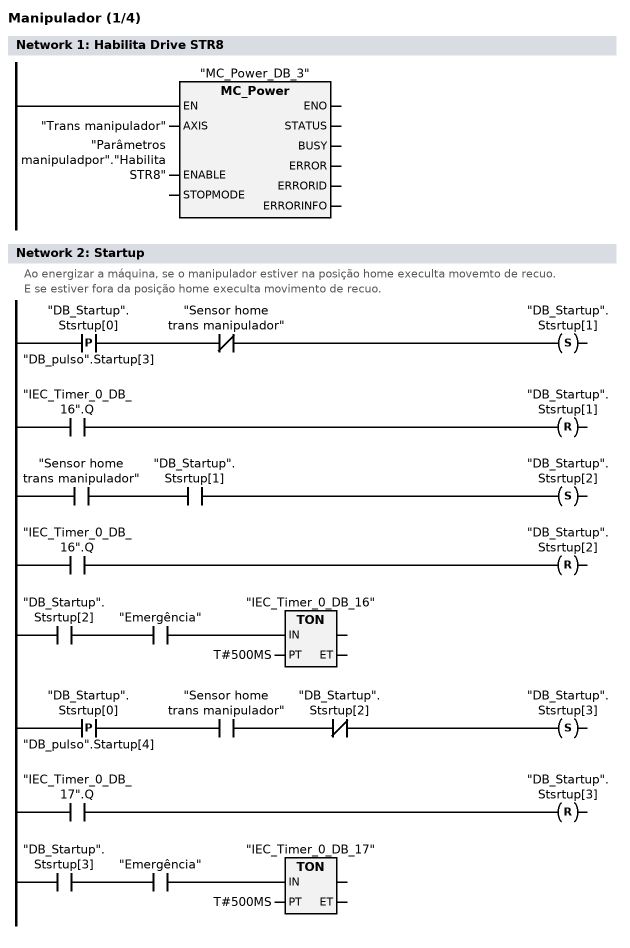
   "MC_Power_DB_3"(Axis := "Trans manipulador", Enable := "Parâmetros manipuladpor"."Habilita STR8");   // MC_Power
END_REGION

REGION Network 2: Startup
   // Ao energizar a máquina, se o manipulador estiver na posição home execulta movemto de recuo.
   // E se estiver fora da posição home execulta movimento de recuo.
   #_w1 := "DB_Startup".Stsrtup[0] AND NOT "DB_pulso".Startup[3];   // rising edge of "DB_Startup".Stsrtup[0]
   "DB_pulso".Startup[3] := "DB_Startup".Stsrtup[0];
   IF #_w1 AND NOT "Sensor home trans manipulador" THEN "DB_Startup".Stsrtup[1] := TRUE; END_IF;
   IF "IEC_Timer_0_DB_16".Q THEN "DB_Startup".Stsrtup[1] := FALSE; END_IF;
   IF "Sensor home trans manipulador" AND "DB_Startup".Stsrtup[1] THEN
       "DB_Startup".Stsrtup[2] := TRUE;
   END_IF;
   IF "IEC_Timer_0_DB_16".Q THEN "DB_Startup".Stsrtup[2] := FALSE; END_IF;
   "IEC_Timer_0_DB_16".TON(IN := "DB_Startup".Stsrtup[2] AND "Emergência", PT := T#500MS);
   #_w2 := "DB_Startup".Stsrtup[0] AND NOT "DB_pulso".Startup[4];   // rising edge of "DB_Startup".Stsrtup[0]
   "DB_pulso".Startup[4] := "DB_Startup".Stsrtup[0];
   IF #_w2 AND "Sensor home trans manipulador" AND NOT "DB_Startup".Stsrtup[2] THEN
       "DB_Startup".Stsrtup[3] := TRUE;
   END_IF;
   IF "IEC_Timer_0_DB_17".Q THEN "DB_Startup".Stsrtup[3] := FALSE; END_IF;
   "IEC_Timer_0_DB_17".TON(IN := "DB_Startup".Stsrtup[3] AND "Emergência", PT := T#500MS);
END_REGION

REGION Network 3: Home manipulador
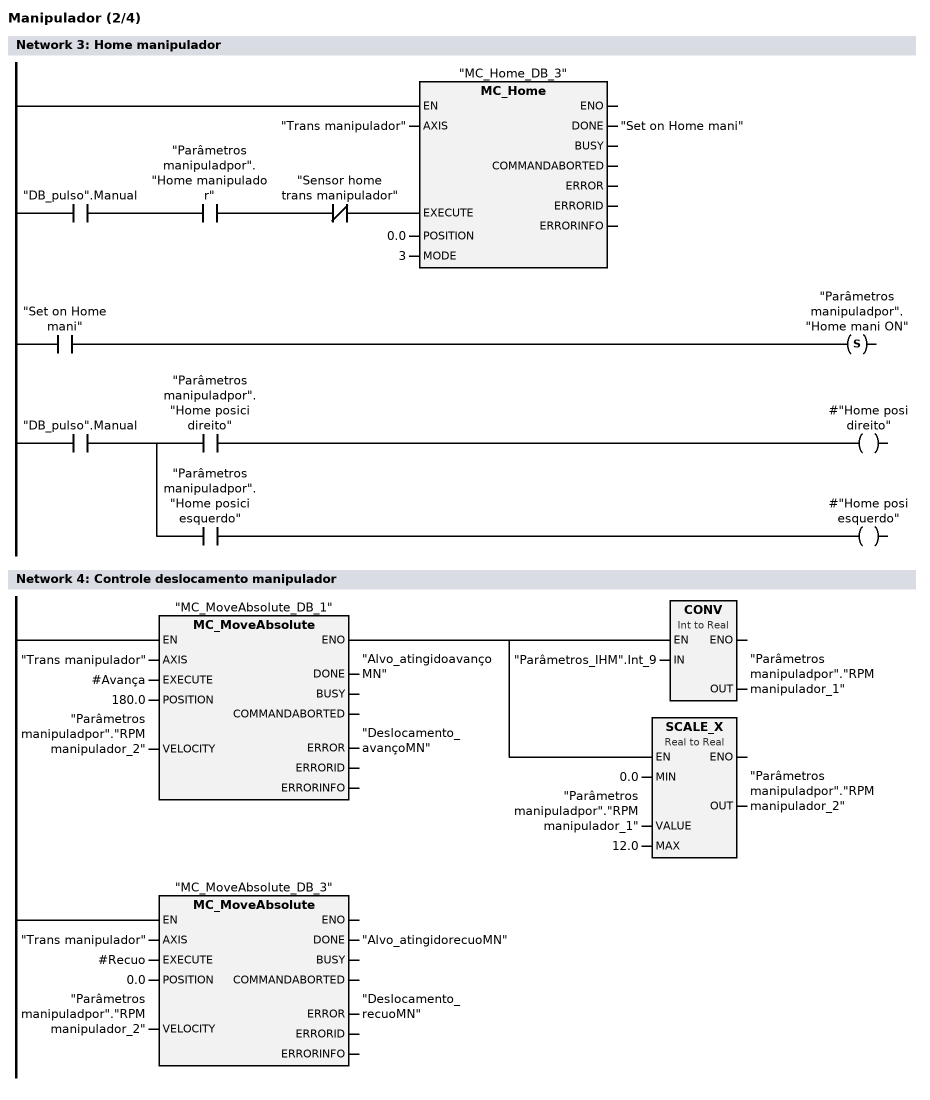
   "MC_Home_DB_3"(Axis := "Trans manipulador",   // MC_Home
                  Execute := "DB_pulso".Manual AND "Parâmetros manipuladpor"."Home manipulador" AND NOT "Sensor home trans manipulador",
                  Position := 0.0,
                  Mode := 3,
                  Done => "Set on Home mani");
   IF "Set on Home mani" THEN "Parâmetros manipuladpor"."Home mani ON" := TRUE; END_IF;
   #"Home posi direito" := "DB_pulso".Manual AND "Parâmetros manipuladpor"."Home posici direito";
   #"Home posi esquerdo" := "DB_pulso".Manual AND "Parâmetros manipuladpor"."Home posici esquerdo";
END_REGION

REGION Network 4: Controle deslocamento manipulador
   // ENO of a box is taken as its EN; it also drops when the box reports an error
   "MC_MoveAbsolute_DB_1"(Axis := "Trans manipulador",   // MC_MoveAbsolute
                          Execute := #Avança,
                          Position := 180.0,
                          Velocity := "Parâmetros manipuladpor"."RPM manipulador_2",
                          Done => "Alvo_atingidoavançoMN",
                          Error => "Deslocamento_avançoMN");
   "Parâmetros manipuladpor"."RPM manipulador_1" := INT_TO_REAL("Parâmetros_IHM".Int_9);
   "Parâmetros manipuladpor"."RPM manipulador_2" := SCALE_X(MIN := 0.0, VALUE := "Parâmetros manipuladpor"."RPM manipulador_1", MAX := 12.0);
   "MC_MoveAbsolute_DB_3"(Axis := "Trans manipulador",   // MC_MoveAbsolute
                          Execute := #Recuo,
                          Position := 0.0,
                          Velocity := "Parâmetros manipuladpor"."RPM manipulador_2",
                          Done => "Alvo_atingidorecuoMN",
                          Error => "Deslocamento_recuoMN");
END_REGION

REGION Network 5: Controle manual avanço recuo manipulador
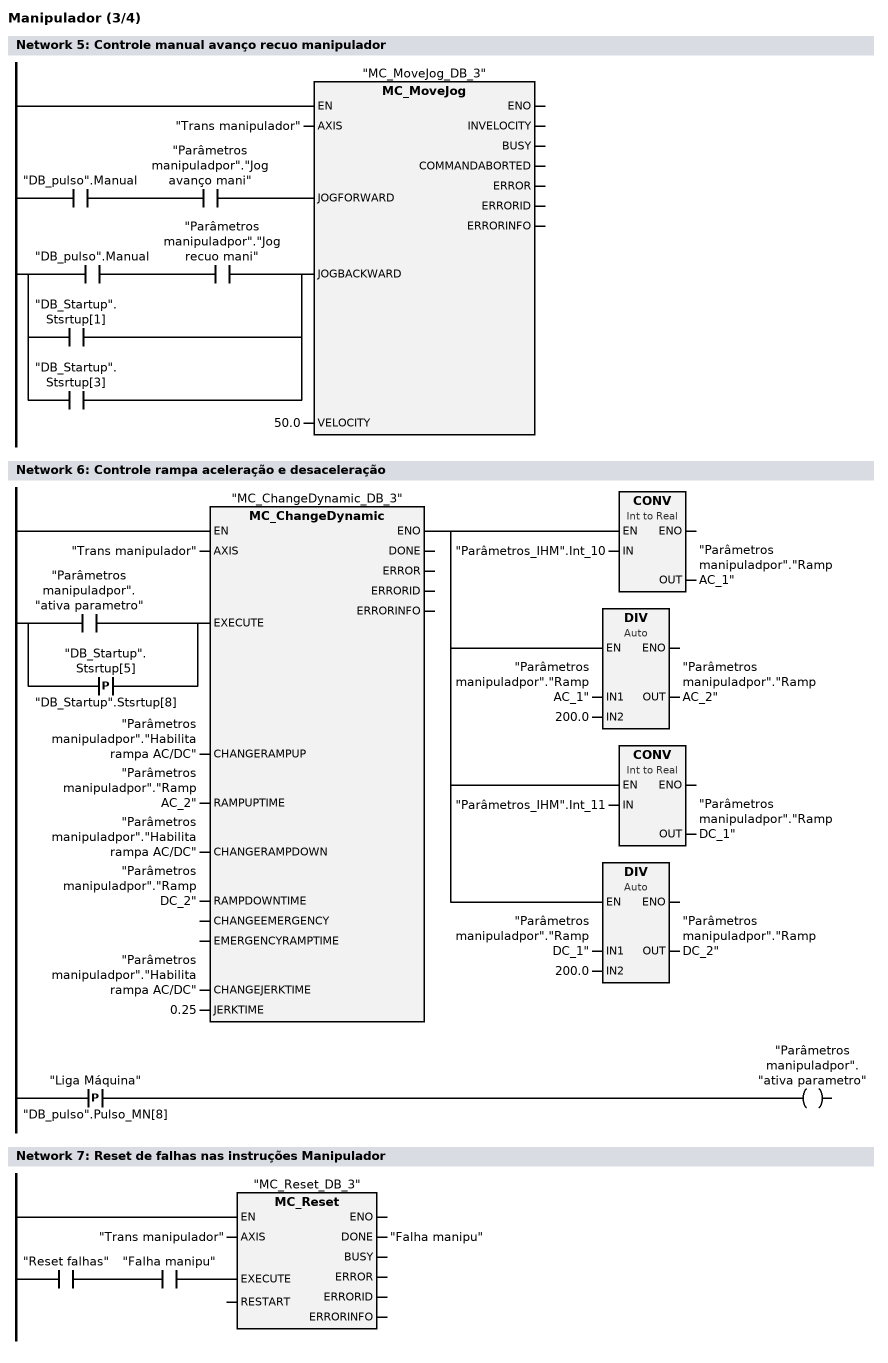
   "MC_MoveJog_DB_3"(Axis := "Trans manipulador",   // MC_MoveJog
                     JogForward := "DB_pulso".Manual AND "Parâmetros manipuladpor"."Jog avanço mani",
                     JogBackward := ("DB_pulso".Manual AND "Parâmetros manipuladpor"."Jog recuo mani") OR "DB_Startup".Stsrtup[1] OR "DB_Startup".Stsrtup[3],
                     Velocity := 50.0);
END_REGION

REGION Network 6: Controle rampa aceleração e desaceleração
   // ENO of a box is taken as its EN; it also drops when the box reports an error
   #_w1 := "DB_Startup".Stsrtup[5] AND NOT "DB_Startup".Stsrtup[8];   // rising edge of "DB_Startup".Stsrtup[5]
   "DB_Startup".Stsrtup[8] := "DB_Startup".Stsrtup[5];
   "MC_ChangeDynamic_DB_3"(Axis := "Trans manipulador",   // MC_ChangeDynamic
                           Execute := "Parâmetros manipuladpor"."ativa parametro" OR #_w1,
                           ChangeRampUp := "Parâmetros manipuladpor"."Habilita rampa AC/DC",
                           RampUpTime := "Parâmetros manipuladpor"."Ramp AC_2",
                           ChangeRampDown := "Parâmetros manipuladpor"."Habilita rampa AC/DC",
                           RampDownTime := "Parâmetros manipuladpor"."Ramp DC_2",
                           ChangeJerkTime := "Parâmetros manipuladpor"."Habilita rampa AC/DC",
                           JerkTime := 0.25);
   "Parâmetros manipuladpor"."Ramp AC_1" := INT_TO_REAL("Parâmetros_IHM".Int_10);
   "Parâmetros manipuladpor"."Ramp AC_2" := "Parâmetros manipuladpor"."Ramp AC_1" / 200.0;
   "Parâmetros manipuladpor"."Ramp DC_1" := INT_TO_REAL("Parâmetros_IHM".Int_11);
   "Parâmetros manipuladpor"."Ramp DC_2" := "Parâmetros manipuladpor"."Ramp DC_1" / 200.0;
   #_w2 := "Liga Máquina" AND NOT "DB_pulso".Pulso_MN[8];   // rising edge of "Liga Máquina"
   "DB_pulso".Pulso_MN[8] := "Liga Máquina";
   "Parâmetros manipuladpor"."ativa parametro" := #_w2;
END_REGION

REGION Network 7: Reset de falhas nas instruções Manipulador
   "MC_Reset_DB_3"(Axis := "Trans manipulador",   // MC_Reset
                   Execute := "Reset falhas" AND "Falha manipu",
                   Done => "Falha manipu");
END_REGION

REGION Network 8
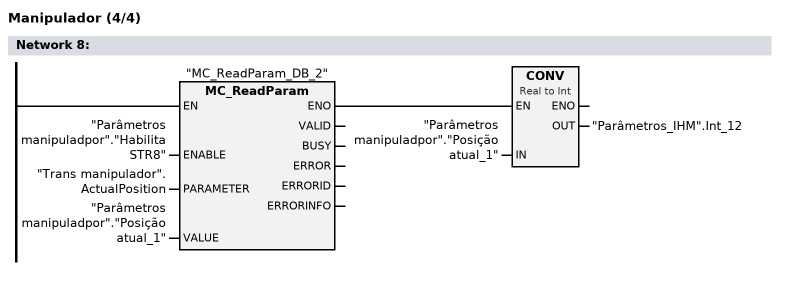
   // ENO of a box is taken as its EN; it also drops when the box reports an error
   "MC_ReadParam_DB_2"(Enable := "Parâmetros manipuladpor"."Habilita STR8",   // MC_ReadParam
                       Parameter := "Trans manipulador".ActualPosition,
                       Value := "Parâmetros manipuladpor"."Posição atual_1");
   "Parâmetros_IHM".Int_12 := REAL_TO_INT("Parâmetros manipuladpor"."Posição atual_1");
END_REGION
END_FUNCTION

FUNCTION "Came" : Void   // FC5, LAD
{ S7_Optimized_Access := 'TRUE' }
VERSION : 0.1
   VAR_INPUT
      Pos_Atual : Int;
      Pos_Start : Int;
      Pos_Stop : Int;
   END_VAR
   VAR_IN_OUT
      Pulso_came : Bool;
      Came : Bool;
   END_VAR
   VAR_TEMP   // added for the SCL form of the ladder/FBD networks
      _w1 : Bool;
   END_VAR
BEGIN

REGION Network 1
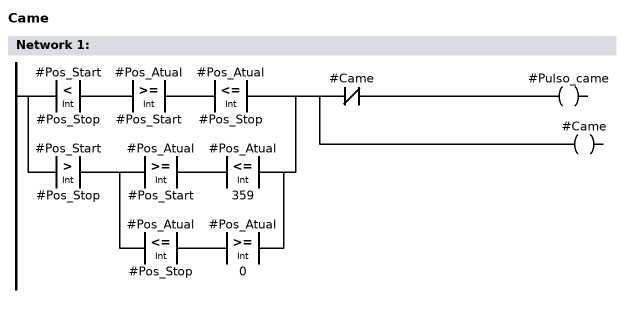
   RUNG wire#powerrail
      { S7_Templates := "SrcType := Int" } LT_Contact(in1 := #Pos_Start, in2 := #Pos_Stop)
      { S7_Templates := "SrcType := Int" } GE_Contact(in1 := #Pos_Atual, in2 := #Pos_Start)
      { S7_Templates := "SrcType := Int" } LE_Contact(in1 := #Pos_Atual, in2 := #Pos_Stop)
      wire#w1
      I_Contact( #Came )
      Coil( #Pulso_came )
   END_RUNG
   RUNG wire#powerrail
      { S7_Templates := "SrcType := Int" } GT_Contact(in1 := #Pos_Start, in2 := #Pos_Stop)
      wire#w2
      { S7_Templates := "SrcType := Int" } GE_Contact(in1 := #Pos_Atual, in2 := #Pos_Start)
      { S7_Templates := "SrcType := Int" } LE_Contact(in1 := #Pos_Atual, in2 := 359)
   END_RUNG wire#w1
   RUNG wire#w2
      { S7_Templates := "SrcType := Int" } LE_Contact(in1 := #Pos_Atual, in2 := #Pos_Stop)
      { S7_Templates := "SrcType := Int" } GE_Contact(in1 := #Pos_Atual, in2 := 0)
   END_RUNG wire#w1
   RUNG wire#w1
      Coil( #Came )
   END_RUNG
   // the same network as SCL:
   #_w1 := ((#Pos_Start < #Pos_Stop) AND (#Pos_Atual >= #Pos_Start) AND (#Pos_Atual <= #Pos_Stop)) OR ((#Pos_Start > #Pos_Stop) AND (((#Pos_Atual >= #Pos_Start) AND (#Pos_Atual <= 359)) OR ((#Pos_Atual <= #Pos_Stop) AND (#Pos_Atual >= 0))));
   #Pulso_came := #_w1 AND NOT #Came;
   #Came := #_w1;
END_REGION
END_FUNCTION

FUNCTION "Alimentador de frasco e tampa" : Void   // FC6, LAD
{ S7_Optimized_Access := 'TRUE' }
VERSION : 0.1
   VAR_TEMP   // added for the SCL form of the ladder/FBD networks
      _w1 : Bool;
      _w2 : Bool;
      _w3 : Bool;
      _w4 : Bool;
      _w5 : Bool;
      _w6 : Bool;
      _w7 : Bool;
      _w8 : Bool;
   END_VAR
BEGIN

REGION Network 1: Liga desliga alimentadores
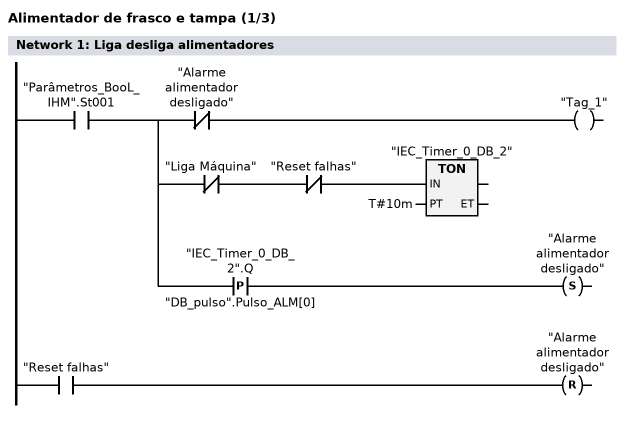
   "Tag_1" := "Parâmetros_BooL_IHM".St001 AND NOT "Alarme alimentador desligado";
   "IEC_Timer_0_DB_2".TON(IN := "Parâmetros_BooL_IHM".St001 AND NOT "Liga Máquina" AND NOT "Reset falhas",
                          PT := T#10m);
   #_w1 := "Parâmetros_BooL_IHM".St001 AND "IEC_Timer_0_DB_2".Q AND NOT "DB_pulso".Pulso_ALM[0];   // rising edge of "IEC_Timer_0_DB_2".Q
   "DB_pulso".Pulso_ALM[0] := "IEC_Timer_0_DB_2".Q;
   IF #_w1 THEN "Alarme alimentador desligado" := TRUE; END_IF;
   IF "Reset falhas" THEN "Alarme alimentador desligado" := FALSE; END_IF;
END_REGION

REGION Network 2: Controle de alimentação panela vibratória frasco
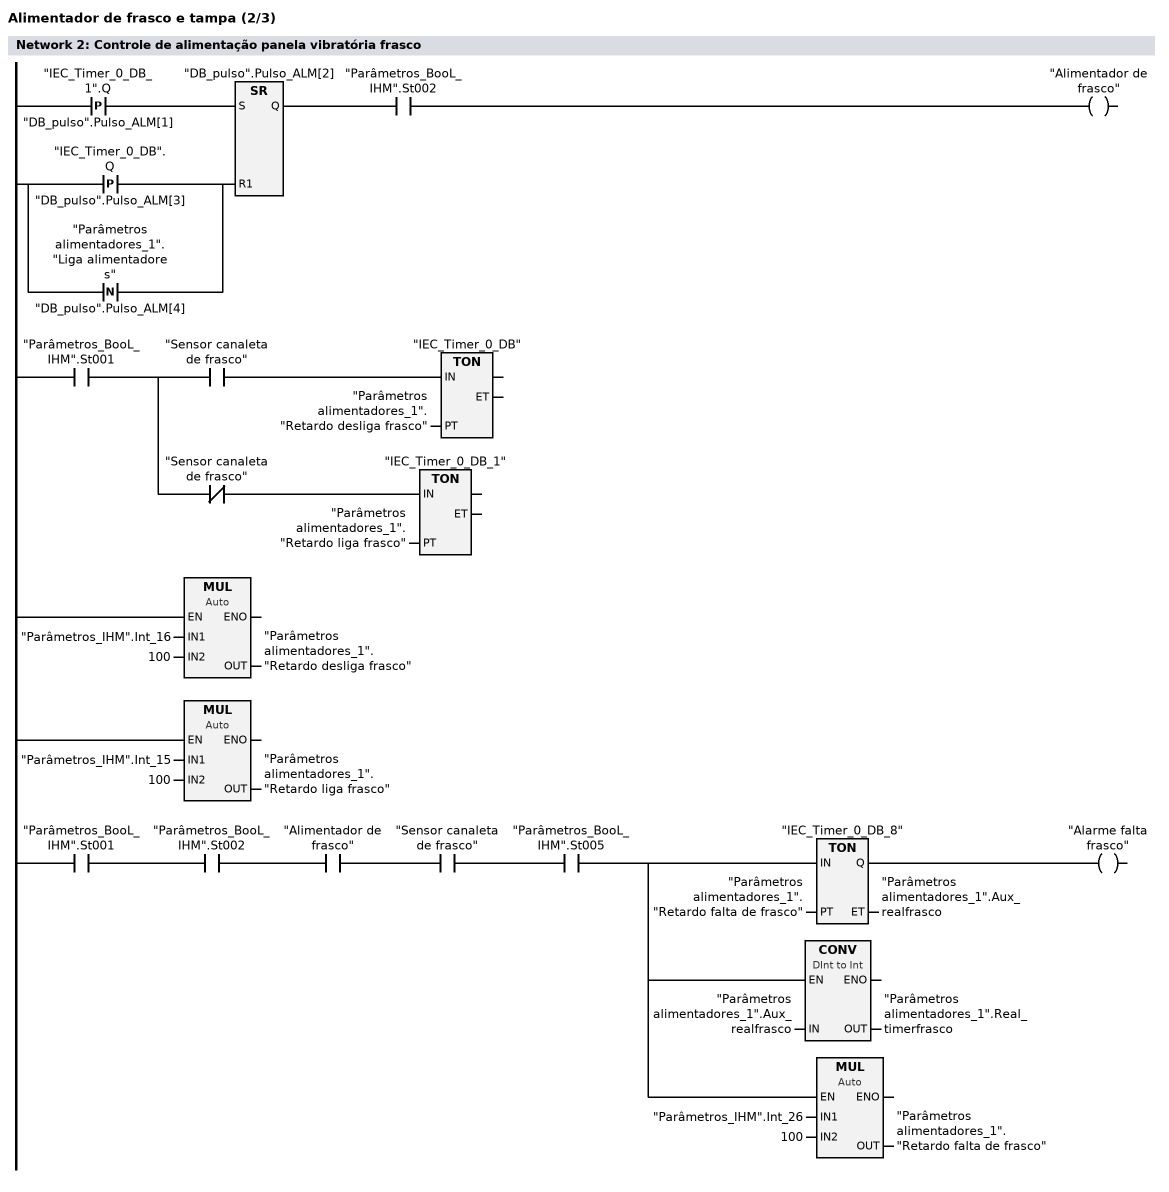
   #_w1 := "IEC_Timer_0_DB_1".Q AND NOT "DB_pulso".Pulso_ALM[1];   // rising edge of "IEC_Timer_0_DB_1".Q
   "DB_pulso".Pulso_ALM[1] := "IEC_Timer_0_DB_1".Q;
   #_w2 := "IEC_Timer_0_DB".Q AND NOT "DB_pulso".Pulso_ALM[3];   // rising edge of "IEC_Timer_0_DB".Q
   "DB_pulso".Pulso_ALM[3] := "IEC_Timer_0_DB".Q;
   #_w3 := NOT "Parâmetros alimentadores_1"."Liga alimentadores" AND "DB_pulso".Pulso_ALM[4];   // falling edge of "Parâmetros alimentadores_1"."Liga alimentadores"
   "DB_pulso".Pulso_ALM[4] := "Parâmetros alimentadores_1"."Liga alimentadores";
   IF #_w1 THEN
       "DB_pulso".Pulso_ALM[2] := TRUE;   // SR flip-flop
   END_IF;
   IF #_w2 OR #_w3 THEN "DB_pulso".Pulso_ALM[2] := FALSE; END_IF;
   "Alimentador de frasco" := "DB_pulso".Pulso_ALM[2] AND "Parâmetros_BooL_IHM".St002;
   "IEC_Timer_0_DB".TON(IN := "Parâmetros_BooL_IHM".St001 AND "Sensor canaleta de frasco",
                        PT := "Parâmetros alimentadores_1"."Retardo desliga frasco");
   "IEC_Timer_0_DB_1".TON(IN := "Parâmetros_BooL_IHM".St001 AND NOT "Sensor canaleta de frasco",
                          PT := "Parâmetros alimentadores_1"."Retardo liga frasco");
   "Parâmetros alimentadores_1"."Retardo desliga frasco" := "Parâmetros_IHM".Int_16 * 100;
   "Parâmetros alimentadores_1"."Retardo liga frasco" := "Parâmetros_IHM".Int_15 * 100;
   #_w4 := "Parâmetros_BooL_IHM".St001 AND "Parâmetros_BooL_IHM".St002 AND "Alimentador de frasco" AND "Sensor canaleta de frasco" AND "Parâmetros_BooL_IHM".St005;
   "IEC_Timer_0_DB_8".TON(IN := #_w4,
                          PT := "Parâmetros alimentadores_1"."Retardo falta de frasco",
                          ET => "Parâmetros alimentadores_1".Aux_realfrasco);
   "Alarme falta frasco" := "IEC_Timer_0_DB_8".Q;
   IF #_w4 THEN
       "Parâmetros alimentadores_1".Real_timerfrasco := DINT_TO_INT("Parâmetros alimentadores_1".Aux_realfrasco);
       "Parâmetros alimentadores_1"."Retardo falta de frasco" := "Parâmetros_IHM".Int_26 * 100;
   END_IF;
END_REGION

REGION Network 3: Controle de alimentação panela vibratória tampa
